(* IEC 61131-3 sources: CodesysTest/export (part 3) *)

(* ---- FB_PneuBagOpenFingersWithSensorsOLD.st ---- *)
{attribute 'FBVisuCreator'}
FUNCTION_BLOCK FB_PneuBagOpenFingersWithSensorsOLD EXTENDS FB_BaseBagOpenFingersOLD
VAR_INPUT
	fingerActuators : IUpDown;
END_VAR
VAR_OUTPUT
END_VAR
VAR
	bagMissingLeft : BOOL;
	bagMissingRight : BOOL;
	simBagPresentLeft : FB_SimulatedFeedbackPhysicalInput(name := CONCAT(_prefix,'Bag Present Left')) := (minDelay := 20, maxDelay := 30);
	simBagPresentRight : FB_SimulatedFeedbackPhysicalInput(name := CONCAT(_prefix,'Bag Present Right')) := (minDelay := 20, maxDelay := 30);
END_VAR
VAR_IN_OUT
	BagPresentSensorLeft : FB_PhysicalDigitalInput;
	BagPresentSensorRight : FB_PhysicalDigitalInput;
END_VAR

SUPER^();
IF simulateIO THEN
	//RotateDownCMD.simulate := RotateUpCMD.simulate := BagPresentSensorLeft.simulate := BagPresentSensorRight.simulate := TRUE;
	BagPresentSensorLeft.simulate := BagPresentSensorRight.simulate := TRUE;
	EnableSimulation(device := fingerActuators, enableSim := TRUE);
END_IF

simBagPresentLeft(in := fingerActuators.DownAsserted,
					simFeedbackFault := UN00_Globals.simFaults.failedToGrabBagLeftFinger OR UN00_Globals.simFaults.failedToGrabBagBothFingers,
					inputToSimulate := BagPresentSensorLeft);
simBagPresentRight(in := fingerActuators.DownAsserted,
					simFeedbackFault := UN00_Globals.simFaults.failedToGrabBagRightFinger OR UN00_Globals.simFaults.failedToGrabBagBothFingers,
					inputToSimulate := BagPresentSensorRight);

bagMissingLeft := NOT BagPresentSensorLeft.Active;
bagMissingRight := NOT BagPresentSensorRight.Active;

IF delayToGrab.Q THEN
	fingerActuators.MoveDown();
	_bagMissed := (bagMissingLeft OR bagMissingRight) AND delayToCheckBagPresent.Q;
	_bagGrabbed := (BagPresentSensorLeft.Active AND BagPresentSensorRight.Active) AND delayToCheckBagPresent.Q;
	//_grabBagRequest := FALSE;
END_IF

IF _releaseBagRequest THEN
	fingerActuators.MoveUp();
	_releaseBagRequest := FALSE;
	_grabBagRequest := FALSE;
END_IF

METHOD RemovePower
VAR_INPUT
END_VAR

SUPER^.RemovePower();

// Try to exhaust the BOF actuators, if the solenoid valve doesn't have that ability then move the fingers up
IF NOT ExhaustIfPossible(fingerActuators) THEN
	fingerActuators.MoveUp();
END_IF

{attribute 'FBVisuCreator'}
FUNCTION_BLOCK FB_PneuBagOpenFingersWithSensorsOLD EXTENDS FB_BaseBagOpenFingersOLD
VAR_INPUT
	fingerActuators : IUpDown;
END_VAR
VAR_OUTPUT
END_VAR
VAR
	bagMissingLeft : BOOL;
	bagMissingRight : BOOL;
	simBagPresentLeft : FB_SimulatedFeedbackPhysicalInput(name := CONCAT(_prefix,'Bag Present Left')) := (minDelay := 20, maxDelay := 30);
	simBagPresentRight : FB_SimulatedFeedbackPhysicalInput(name := CONCAT(_prefix,'Bag Present Right')) := (minDelay := 20, maxDelay := 30);
END_VAR
VAR_IN_OUT
	BagPresentSensorLeft : FB_PhysicalDigitalInput;
	BagPresentSensorRight : FB_PhysicalDigitalInput;
END_VAR

SUPER^();
IF simulateIO THEN
	//RotateDownCMD.simulate := RotateUpCMD.simulate := BagPresentSensorLeft.simulate := BagPresentSensorRight.simulate := TRUE;
	BagPresentSensorLeft.simulate := BagPresentSensorRight.simulate := TRUE;
	EnableSimulation(device := fingerActuators, enableSim := TRUE);
END_IF

simBagPresentLeft(in := fingerActuators.DownAsserted,
					simFeedbackFault := UN00_Globals.simFaults.failedToGrabBagLeftFinger OR UN00_Globals.simFaults.failedToGrabBagBothFingers,
					inputToSimulate := BagPresentSensorLeft);
simBagPresentRight(in := fingerActuators.DownAsserted,
					simFeedbackFault := UN00_Globals.simFaults.failedToGrabBagRightFinger OR UN00_Globals.simFaults.failedToGrabBagBothFingers,
					inputToSimulate := BagPresentSensorRight);

bagMissingLeft := NOT BagPresentSensorLeft.Active;
bagMissingRight := NOT BagPresentSensorRight.Active;

IF delayToGrab.Q THEN
	fingerActuators.MoveDown();
	_bagMissed := (bagMissingLeft OR bagMissingRight) AND delayToCheckBagPresent.Q;
	_bagGrabbed := (BagPresentSensorLeft.Active AND BagPresentSensorRight.Active) AND delayToCheckBagPresent.Q;
	//_grabBagRequest := FALSE;
END_IF

IF _releaseBagRequest THEN
	fingerActuators.MoveUp();
	_releaseBagRequest := FALSE;
	_grabBagRequest := FALSE;
END_IF

METHOD RemovePower
VAR_INPUT
END_VAR

SUPER^.RemovePower();

// Try to exhaust the BOF actuators, if the solenoid valve doesn't have that ability then move the fingers up
IF NOT ExhaustIfPossible(fingerActuators) THEN
	fingerActuators.MoveUp();
END_IF

(* ---- FB_PneumaticActuator.st ---- *)
FUNCTION_BLOCK FB_PneumaticActuator EXTENDS FB_SolenoidValve IMPLEMENTS ICylinder
VAR_INPUT

END_VAR
VAR_OUTPUT
END_VAR
VAR
	_extendAsserted : BOOL;
	_isExtended : BOOL;
	_retractAsserted : BOOL;
	_isRetracted : BOOL;
END_VAR

PROPERTY ExtendAsserted : BOOL

PROPERTY IsExtended : BOOL

PROPERTY IsRetracted : BOOL

PROPERTY RetractAsserted : BOOL

METHOD Extend

_extendAsserted := TRUE;
_retractAsserted := FALSE;

METHOD Retract

_extendAsserted := FALSE;
_retractAsserted := TRUE;

FUNCTION_BLOCK FB_PneumaticActuator EXTENDS FB_SolenoidValve IMPLEMENTS ICylinder
VAR_INPUT

END_VAR
VAR_OUTPUT
END_VAR
VAR
	_extendAsserted : BOOL;
	_isExtended : BOOL;
	_retractAsserted : BOOL;
	_isRetracted : BOOL;
END_VAR

PROPERTY ExtendAsserted : BOOL

PROPERTY IsExtended : BOOL

PROPERTY IsRetracted : BOOL

PROPERTY RetractAsserted : BOOL

METHOD Extend

_extendAsserted := TRUE;
_retractAsserted := FALSE;

METHOD Retract

_extendAsserted := FALSE;
_retractAsserted := TRUE;

(* ---- FB_PneumaticActuator_UnitTests.st ---- *)
(*
*)
{attribute 'test' := 'multitest'}
{attribute 'testcasename':='Base Pneumatic Actuator/Valve'}
{attribute 'testcategory':='Solenoids'}
{attribute 'testcasetimeout':='15000'}
FUNCTION_BLOCK FB_PneumaticActuator_UnitTests EXTENDS CBM.EtrigA
VAR_INPUT
	xGetTestInfo : BOOL;
    diTestCaseIndex : DINT;
END_VAR
VAR_OUTPUT
    sTestCaseName : STRING;
	sTestCaseCategories : STRING;
    diTestCaseCount : DINT;
    diTestCaseTimeout : DINT;
    sInfo : STRING;
	eError : UnitTestErrors;
    sError : STRING;
    eFailureMode : TM.FAILUREMODE;
END_VAR
VAR
	testee : FB_PneumaticActuator(name := 'Unit Test Actuator');
END_VAR
SUPER^();

{attribute 'hide'}
METHOD prvAbort : BOOL

SUPER^.prvAbort();

xAbortInProgress := FALSE;

{attribute 'hide'}
METHOD prvCyclicAction : BOOL

SUPER^.prvCyclicAction();
THIS^.diTestCaseCount := 3;

CASE diTestCaseIndex OF
    0: // Test Case #0
        IF THIS^.xGetTestInfo THEN
            THIS^.sTestCaseName := 'Step 1: Test Initialzed No State';
            THIS^.sTestCaseCategories := 'Solenoids';
            THIS^.diTestCaseTimeout := 3000;
			xDone := TRUE;
		ELSE
			IF NOT testee.ExtendAsserted
				AND NOT testee.RetractAsserted
				AND NOT testee.IsExtended
				AND NOT testee.IsRetracted
				THEN
				 xDone := TRUE;
			ELSE
				THIS^.sError := 'Initialzed with state (Extended or Retracted)';
				xError := TRUE;
				eError := UnitTestErrors.Failure;
            	eFailureMode := TM.FAILUREMODE.AbortTestCase;
                iError := 1;
			END_IF
        END_IF
    1: // Test Case #1
        IF THIS^.xGetTestInfo THEN
            THIS^.sTestCaseName := 'Step 2: Extend Cylinder';
            THIS^.sTestCaseCategories := 'Solenoids';
            THIS^.diTestCaseTimeout := 3000;
            xDone := TRUE;
		ELSE
			testee.Extend();
			testee.IsExtended := TRUE;
			IF testee.ExtendAsserted
				AND testee.IsExtended
				AND NOT testee.RetractAsserted
				AND NOT testee.IsRetracted
				THEN
				 xDone := TRUE;
			ELSE
				THIS^.sError := 'Failed to extend';
				xError := TRUE;
				eError := UnitTestErrors.Failure;
            	eFailureMode := TM.FAILUREMODE.AbortTestCase;
                iError := 2;
			END_IF
       END_IF

	2:	//
		IF THIS^.xGetTestInfo THEN
            THIS^.sTestCaseName := 'Step 3: Retract Cylinder';
            THIS^.sTestCaseCategories := 'Solenoids';
            THIS^.diTestCaseTimeout := 3000;
            xDone := TRUE;
		ELSE
			testee.Retract();
			testee.IsRetracted := TRUE;
			testee.IsExtended := FALSE;
			IF NOT testee.ExtendAsserted
				AND NOT testee.IsExtended
				AND testee.RetractAsserted
				AND testee.IsRetracted
				THEN
				 xDone := TRUE;
			ELSE
				THIS^.sError := 'Failed to retract';
				xError := TRUE;
				eError := UnitTestErrors.Failure;
            	eFailureMode := TM.FAILUREMODE.AbortTestCase;
                iError := 3;
			END_IF
       END_IF
    ELSE
        IF THIS^.diTestCaseIndex < 0 THEN
            THIS^.diTestCaseCount := 3;
            xDone := TRUE;
        ELSE
            THIS^.sInfo := 'Invalid test case index';
            eError := UnitTestErrors.Failure;
			xError := TRUE;
        END_IF
END_CASE

{attribute 'hide'}
METHOD prvResetOutputs : BOOL

SUPER^.prvResetOutputs();

sTestCaseName := '';
sTestCaseCategories := '';
diTestCaseCount := 0;
diTestCaseTimeout := 0;
sInfo := '';
sError := '';
eFailureMode := TM.FAILUREMODE.AbortTestCase;

{attribute 'hide'}
METHOD prvStart : BOOL

SUPER^.prvStart();

(*
*)
{attribute 'test' := 'multitest'}
{attribute 'testcasename':='Base Pneumatic Actuator/Valve'}
{attribute 'testcategory':='Solenoids'}
{attribute 'testcasetimeout':='15000'}
FUNCTION_BLOCK FB_PneumaticActuator_UnitTests EXTENDS CBM.EtrigA
VAR_INPUT
	xGetTestInfo : BOOL;
    diTestCaseIndex : DINT;
END_VAR
VAR_OUTPUT
    sTestCaseName : STRING;
	sTestCaseCategories : STRING;
    diTestCaseCount : DINT;
    diTestCaseTimeout : DINT;
    sInfo : STRING;
	eError : UnitTestErrors;
    sError : STRING;
    eFailureMode : TM.FAILUREMODE;
END_VAR
VAR
	testee : FB_PneumaticActuator(name := 'Unit Test Actuator');
END_VAR
SUPER^();

{attribute 'hide'}
METHOD prvAbort : BOOL

SUPER^.prvAbort();

xAbortInProgress := FALSE;

{attribute 'hide'}
METHOD prvCyclicAction : BOOL

SUPER^.prvCyclicAction();
THIS^.diTestCaseCount := 3;

CASE diTestCaseIndex OF
    0: // Test Case #0
        IF THIS^.xGetTestInfo THEN
            THIS^.sTestCaseName := 'Step 1: Test Initialzed No State';
            THIS^.sTestCaseCategories := 'Solenoids';
            THIS^.diTestCaseTimeout := 3000;
			xDone := TRUE;
		ELSE
			IF NOT testee.ExtendAsserted
				AND NOT testee.RetractAsserted
				AND NOT testee.IsExtended
				AND NOT testee.IsRetracted
				THEN
				 xDone := TRUE;
			ELSE
				THIS^.sError := 'Initialzed with state (Extended or Retracted)';
				xError := TRUE;
				eError := UnitTestErrors.Failure;
            	eFailureMode := TM.FAILUREMODE.AbortTestCase;
                iError := 1;
			END_IF
        END_IF
    1: // Test Case #1
        IF THIS^.xGetTestInfo THEN
            THIS^.sTestCaseName := 'Step 2: Extend Cylinder';
            THIS^.sTestCaseCategories := 'Solenoids';
            THIS^.diTestCaseTimeout := 3000;
            xDone := TRUE;
		ELSE
			testee.Extend();
			testee.IsExtended := TRUE;
			IF testee.ExtendAsserted
				AND testee.IsExtended
				AND NOT testee.RetractAsserted
				AND NOT testee.IsRetracted
				THEN
				 xDone := TRUE;
			ELSE
				THIS^.sError := 'Failed to extend';
				xError := TRUE;
				eError := UnitTestErrors.Failure;
            	eFailureMode := TM.FAILUREMODE.AbortTestCase;
                iError := 2;
			END_IF
       END_IF

	2:	//
		IF THIS^.xGetTestInfo THEN
            THIS^.sTestCaseName := 'Step 3: Retract Cylinder';
            THIS^.sTestCaseCategories := 'Solenoids';
            THIS^.diTestCaseTimeout := 3000;
            xDone := TRUE;
		ELSE
			testee.Retract();
			testee.IsRetracted := TRUE;
			testee.IsExtended := FALSE;
			IF NOT testee.ExtendAsserted
				AND NOT testee.IsExtended
				AND testee.RetractAsserted
				AND testee.IsRetracted
				THEN
				 xDone := TRUE;
			ELSE
				THIS^.sError := 'Failed to retract';
				xError := TRUE;
				eError := UnitTestErrors.Failure;
            	eFailureMode := TM.FAILUREMODE.AbortTestCase;
                iError := 3;
			END_IF
       END_IF
    ELSE
        IF THIS^.diTestCaseIndex < 0 THEN
            THIS^.diTestCaseCount := 3;
            xDone := TRUE;
        ELSE
            THIS^.sInfo := 'Invalid test case index';
            eError := UnitTestErrors.Failure;
			xError := TRUE;
        END_IF
END_CASE

{attribute 'hide'}
METHOD prvResetOutputs : BOOL

SUPER^.prvResetOutputs();

sTestCaseName := '';
sTestCaseCategories := '';
diTestCaseCount := 0;
diTestCaseTimeout := 0;
sInfo := '';
sError := '';
eFailureMode := TM.FAILUREMODE.AbortTestCase;

{attribute 'hide'}
METHOD prvStart : BOOL

SUPER^.prvStart();

(* ---- FB_PneumaticSealer.st ---- *)
FUNCTION_BLOCK FINAL FB_PneumaticSealer EXTENDS FB_BasicSealer
VAR_INPUT
	cylinder : ICylinder;
END_VAR
VAR_OUTPUT
END_VAR
VAR

END_VAR

SUPER^();

EnableSimulation(cylinder,simulateIO);

IF sealActive THEN
	cylinder.Extend();
ELSE
	cylinder.Retract();
END_IF

{attribute 'monitoring' := 'variable'}
PROPERTY SealComplete : BOOL

METHOD BeginSealing

_beginSealing := TRUE;
sealTimer.IN := FALSE;
_sealComplete := FALSE;

FUNCTION_BLOCK FINAL FB_PneumaticSealer EXTENDS FB_BasicSealer
VAR_INPUT
	cylinder : ICylinder;
END_VAR
VAR_OUTPUT
END_VAR
VAR

END_VAR

SUPER^();

EnableSimulation(cylinder,simulateIO);

IF sealActive THEN
	cylinder.Extend();
ELSE
	cylinder.Retract();
END_IF

{attribute 'monitoring' := 'variable'}
PROPERTY SealComplete : BOOL

METHOD BeginSealing

_beginSealing := TRUE;
sealTimer.IN := FALSE;
_sealComplete := FALSE;

(* ---- FB_PneumaticVacuumCups.st ---- *)
FUNCTION_BLOCK FB_PneumaticVacuumCups EXTENDS FB_BaseComponent IMPLEMENTS IVacuumBagOpen
VAR_INPUT

END_VAR
VAR_OUTPUT

END_VAR
VAR
	_vacuumOn : BOOL;
END_VAR
VAR_IN_OUT
	vacGenerator : FB_VacuumGenerator;
END_VAR
SUPER^();

{attribute 'monitoring' := 'variable'}
PROPERTY VacuumOn : BOOL

METHOD StartVacuum

vacGenerator.GeneratorsOn();
_vacuumOn := TRUE;

METHOD StopVacuum

vacGenerator.GeneratorsOff();
_vacuumOn := FALSE;

(* ---- FB_PneumaticVacuumCups_UnitTests.st ---- *)
{attribute 'test' := 'multitest'}
{attribute 'testcasename':='Pneumatic Vacuum Cups'}
{attribute 'testcategory':='Machine Components'}
{attribute 'testcasetimeout':='15000'}

FUNCTION_BLOCK FB_PneumaticVacuumCups_UnitTests EXTENDS CBM.EtrigA
VAR_INPUT
	xGetTestInfo : BOOL;
    diTestCaseIndex : DINT;
END_VAR
VAR_OUTPUT
    sTestCaseName : STRING;
	sTestCaseCategories : STRING;
    diTestCaseCount : DINT;
    diTestCaseTimeout : DINT;
    sInfo : STRING;
	eError : UnitTestErrors;
    sError : STRING;
    eFailureMode : TM.FAILUREMODE;
END_VAR
VAR
	testVacGenerator : FB_VacuumGenerator(name := 'Test Vac Generator');
	testee : FB_PneumaticVacuumCups(name := 'Test Pneumatic Vac Cups');
END_VAR
SUPER^();
testVacGenerator();
testee(vacGenerator := testVacGenerator);

{attribute 'hide'}
METHOD prvAbort : BOOL

SUPER^.prvAbort();

xAbortInProgress := FALSE;

{attribute 'hide'}
METHOD prvCyclicAction : BOOL

SUPER^.prvCyclicAction();

CASE diTestCaseIndex OF
    0: 	IF THIS^.xGetTestInfo THEN
            THIS^.sTestCaseName := 'Step 1: Check Vacuum Is Off On Initialze';
            THIS^.sTestCaseCategories := 'General';
            THIS^.diTestCaseTimeout := 3000;
			xDone := TRUE;
		ELSE
			IF testee.VacuumOn = FALSE THEN
				 xDone := TRUE;
			ELSE
				THIS^.sError := 'Vacuum On, should be off on initialize';
				xError := TRUE;
				eError := UnitTestErrors.Failure;
            	eFailureMode := TM.FAILUREMODE.AbortTestCase;
                iError := 1;
			END_IF
        END_IF
    1: 	IF THIS^.xGetTestInfo THEN
            THIS^.sTestCaseName := 'Step 2: Start Vacuum';
            THIS^.sTestCaseCategories := 'General';
            THIS^.diTestCaseTimeout := 3000;
			xDone := TRUE;
		ELSE
			testee.StartVacuum();
			IF testee.VacuumOn AND testVacGenerator.Solenoid0Asserted THEN
				 xDone := TRUE;
			ELSE
				THIS^.sError := 'Vacuum Off, should be on';
				xError := TRUE;
				eError := UnitTestErrors.Failure;
            	eFailureMode := TM.FAILUREMODE.AbortTestCase;
                iError := 1;
			END_IF
        END_IF

	2: 	IF THIS^.xGetTestInfo THEN
            THIS^.sTestCaseName := 'Step 3: Stop Vacuum';
            THIS^.sTestCaseCategories := 'General';
            THIS^.diTestCaseTimeout := 3000;
			xDone := TRUE;
		ELSE
			testee.StopVacuum();
			IF NOT testee.VacuumOn AND NOT testVacGenerator.Solenoid0Asserted THEN
				 xDone := TRUE;
			ELSE
				THIS^.sError := 'Vacumm On, should be off';
				xError := TRUE;
				eError := UnitTestErrors.Failure;
            	eFailureMode := TM.FAILUREMODE.AbortTestCase;
                iError := 1;
			END_IF
        END_IF

   	3: 	IF THIS^.xGetTestInfo THEN
            THIS^.sTestCaseName := 'Step 4: ';
            THIS^.sTestCaseCategories := 'General';
            THIS^.diTestCaseTimeout := 3000;
			xDone := TRUE;
		ELSE
			(*TEST SOMETHING HERE*)
			IF (*CONNDITION*) FALSE THEN
				 xDone := TRUE;
			ELSE
				THIS^.sError := '';
				xError := TRUE;
				eError := UnitTestErrors.Failure;
            	eFailureMode := TM.FAILUREMODE.AbortTestCase;
                iError := 1;
			END_IF
        END_IF

	4: 	IF THIS^.xGetTestInfo THEN
            THIS^.sTestCaseName := 'Step 5: ';
            THIS^.sTestCaseCategories := 'General';
            THIS^.diTestCaseTimeout := 3000;
			xDone := TRUE;
		ELSE
			(*TEST SOMETHING HERE*)
			IF (*CONNDITION*) FALSE THEN
				 xDone := TRUE;
			ELSE
				THIS^.sError := '';
				xError := TRUE;
				eError := UnitTestErrors.Failure;
            	eFailureMode := TM.FAILUREMODE.AbortTestCase;
                iError := 1;
			END_IF
        END_IF

	5: 	IF THIS^.xGetTestInfo THEN
            THIS^.sTestCaseName := 'Step 6: ';
            THIS^.sTestCaseCategories := 'General';
            THIS^.diTestCaseTimeout := 3000;
			xDone := TRUE;
		ELSE
			(*TEST SOMETHING HERE*)
			IF (*CONNDITION*) FALSE THEN
				 xDone := TRUE;
			ELSE
				THIS^.sError := '';
				xError := TRUE;
				eError := UnitTestErrors.Failure;
            	eFailureMode := TM.FAILUREMODE.AbortTestCase;
                iError := 1;
			END_IF
        END_IF

	6: 	IF THIS^.xGetTestInfo THEN
            THIS^.sTestCaseName := 'Step 7: ';
            THIS^.sTestCaseCategories := 'General';
            THIS^.diTestCaseTimeout := 3000;
			xDone := TRUE;
		ELSE
			(*TEST SOMETHING HERE*)
			IF (*CONNDITION*) FALSE THEN
				 xDone := TRUE;
			ELSE
				THIS^.sError := '';
				xError := TRUE;
				eError := UnitTestErrors.Failure;
            	eFailureMode := TM.FAILUREMODE.AbortTestCase;
                iError := 1;
			END_IF
        END_IF
    ELSE
        IF THIS^.diTestCaseIndex < 0 THEN
            THIS^.diTestCaseCount := 3;
            xDone := TRUE;
        ELSE
            THIS^.sInfo := 'Invalid test case index';
            eError := UnitTestErrors.Failure;
			xError := TRUE;
        END_IF
END_CASE

{attribute 'hide'}
METHOD prvResetOutputs : BOOL

SUPER^.prvResetOutputs();

sTestCaseName := '';
sTestCaseCategories := '';
diTestCaseCount := 0;
diTestCaseTimeout := 0;
sInfo := '';
sError := '';
eFailureMode := TM.FAILUREMODE.AbortTestCase;

{attribute 'hide'}
METHOD prvStart : BOOL

{attribute 'test' := 'multitest'}
{attribute 'testcasename':='Pneumatic Vacuum Cups'}
{attribute 'testcategory':='Machine Components'}
{attribute 'testcasetimeout':='15000'}

FUNCTION_BLOCK FB_PneumaticVacuumCups_UnitTests EXTENDS CBM.EtrigA
VAR_INPUT
	xGetTestInfo : BOOL;
    diTestCaseIndex : DINT;
END_VAR
VAR_OUTPUT
    sTestCaseName : STRING;
	sTestCaseCategories : STRING;
    diTestCaseCount : DINT;
    diTestCaseTimeout : DINT;
    sInfo : STRING;
	eError : UnitTestErrors;
    sError : STRING;
    eFailureMode : TM.FAILUREMODE;
END_VAR
VAR
	testVacGenerator : FB_VacuumGenerator(name := 'Test Vac Generator');
	testee : FB_PneumaticVacuumCups(name := 'Test Pneumatic Vac Cups');
END_VAR
SUPER^();
testVacGenerator();
testee(vacGenerator := testVacGenerator);

{attribute 'hide'}
METHOD prvAbort : BOOL

SUPER^.prvAbort();

xAbortInProgress := FALSE;

{attribute 'hide'}
METHOD prvCyclicAction : BOOL

SUPER^.prvCyclicAction();

CASE diTestCaseIndex OF
    0: 	IF THIS^.xGetTestInfo THEN
            THIS^.sTestCaseName := 'Step 1: Check Vacuum Is Off On Initialze';
            THIS^.sTestCaseCategories := 'General';
            THIS^.diTestCaseTimeout := 3000;
			xDone := TRUE;
		ELSE
			IF testee.VacuumOn = FALSE THEN
				 xDone := TRUE;
			ELSE
				THIS^.sError := 'Vacuum On, should be off on initialize';
				xError := TRUE;
				eError := UnitTestErrors.Failure;
            	eFailureMode := TM.FAILUREMODE.AbortTestCase;
                iError := 1;
			END_IF
        END_IF
    1: 	IF THIS^.xGetTestInfo THEN
            THIS^.sTestCaseName := 'Step 2: Start Vacuum';
            THIS^.sTestCaseCategories := 'General';
            THIS^.diTestCaseTimeout := 3000;
			xDone := TRUE;
		ELSE
			testee.StartVacuum();
			IF testee.VacuumOn AND testVacGenerator.Solenoid0Asserted THEN
				 xDone := TRUE;
			ELSE
				THIS^.sError := 'Vacuum Off, should be on';
				xError := TRUE;
				eError := UnitTestErrors.Failure;
            	eFailureMode := TM.FAILUREMODE.AbortTestCase;
                iError := 1;
			END_IF
        END_IF

	2: 	IF THIS^.xGetTestInfo THEN
            THIS^.sTestCaseName := 'Step 3: Stop Vacuum';
            THIS^.sTestCaseCategories := 'General';
            THIS^.diTestCaseTimeout := 3000;
			xDone := TRUE;
		ELSE
			testee.StopVacuum();
			IF NOT testee.VacuumOn AND NOT testVacGenerator.Solenoid0Asserted THEN
				 xDone := TRUE;
			ELSE
				THIS^.sError := 'Vacumm On, should be off';
				xError := TRUE;
				eError := UnitTestErrors.Failure;
            	eFailureMode := TM.FAILUREMODE.AbortTestCase;
                iError := 1;
			END_IF
        END_IF

   	3: 	IF THIS^.xGetTestInfo THEN
            THIS^.sTestCaseName := 'Step 4: ';
            THIS^.sTestCaseCategories := 'General';
            THIS^.diTestCaseTimeout := 3000;
			xDone := TRUE;
		ELSE
			(*TEST SOMETHING HERE*)
			IF (*CONNDITION*) FALSE THEN
				 xDone := TRUE;
			ELSE
				THIS^.sError := '';
				xError := TRUE;
				eError := UnitTestErrors.Failure;
            	eFailureMode := TM.FAILUREMODE.AbortTestCase;
                iError := 1;
			END_IF
        END_IF

	4: 	IF THIS^.xGetTestInfo THEN
            THIS^.sTestCaseName := 'Step 5: ';
            THIS^.sTestCaseCategories := 'General';
            THIS^.diTestCaseTimeout := 3000;
			xDone := TRUE;
		ELSE
			(*TEST SOMETHING HERE*)
			IF (*CONNDITION*) FALSE THEN
				 xDone := TRUE;
			ELSE
				THIS^.sError := '';
				xError := TRUE;
				eError := UnitTestErrors.Failure;
            	eFailureMode := TM.FAILUREMODE.AbortTestCase;
                iError := 1;
			END_IF
        END_IF

	5: 	IF THIS^.xGetTestInfo THEN
            THIS^.sTestCaseName := 'Step 6: ';
            THIS^.sTestCaseCategories := 'General';
            THIS^.diTestCaseTimeout := 3000;
			xDone := TRUE;
		ELSE
			(*TEST SOMETHING HERE*)
			IF (*CONNDITION*) FALSE THEN
				 xDone := TRUE;
			ELSE
				THIS^.sError := '';
				xError := TRUE;
				eError := UnitTestErrors.Failure;
            	eFailureMode := TM.FAILUREMODE.AbortTestCase;
                iError := 1;
			END_IF
        END_IF

	6: 	IF THIS^.xGetTestInfo THEN
            THIS^.sTestCaseName := 'Step 7: ';
            THIS^.sTestCaseCategories := 'General';
            THIS^.diTestCaseTimeout := 3000;
			xDone := TRUE;
		ELSE
			(*TEST SOMETHING HERE*)
			IF (*CONNDITION*) FALSE THEN
				 xDone := TRUE;
			ELSE
				THIS^.sError := '';
				xError := TRUE;
				eError := UnitTestErrors.Failure;
            	eFailureMode := TM.FAILUREMODE.AbortTestCase;
                iError := 1;
			END_IF
        END_IF
    ELSE
        IF THIS^.diTestCaseIndex < 0 THEN
            THIS^.diTestCaseCount := 3;
            xDone := TRUE;
        ELSE
            THIS^.sInfo := 'Invalid test case index';
            eError := UnitTestErrors.Failure;
			xError := TRUE;
        END_IF
END_CASE

{attribute 'hide'}
METHOD prvResetOutputs : BOOL

SUPER^.prvResetOutputs();

sTestCaseName := '';
sTestCaseCategories := '';
diTestCaseCount := 0;
diTestCaseTimeout := 0;
sInfo := '';
sError := '';
eFailureMode := TM.FAILUREMODE.AbortTestCase;

{attribute 'hide'}
METHOD prvStart : BOOL

(* ---- FB_PneumaticVerticalActuator.st ---- *)
FUNCTION_BLOCK FB_PneumaticVerticalActuator EXTENDS FB_PneumaticActuator IMPLEMENTS IUpDown
VAR_INPUT
	cylinder : ICylinder;
END_VAR
VAR_OUTPUT
END_VAR
VAR
END_VAR
VAR_IN_OUT
END_VAR

//	Function Block: FB_PneumaticVerticalActuator
//	Description: Wrapper for a cylinder with Up/Down substitiuted for Extend/Retract
//
//
//	Usage:
//
//	Created by: Ben Hess
//	Created Date: 6-27-2019

EnableSimulation(cylinder, _simulateActive);

PROPERTY UpAsserted : BOOL

PROPERTY DownAsserted : BOOL

PROPERTY IsDown : BOOL

PROPERTY IsUp : BOOL

METHOD MoveDown

cylinder.Extend();

METHOD MoveUp

cylinder.Retract();

(* ---- FB_PneuPBarWithAdjPass.st ---- *)
FUNCTION_BLOCK FB_PneuPBarWithAdjPass EXTENDS FB_BaseComponent IMPLEMENTS IPressureBar, IHomable, IPostHomeMove
VAR_INPUT
	simulateIO : BOOL;												// Simulate all I/O for testing
	passthroughMotor : REFERENCE TO Sharp_Motion.Axis_REF;			// The motor axis for the passthrough
	ptVelo : REAL := 0.5;											// Passthrough Motor Velocity
	ptAccel : REAL := 10.0;											// Passthrough Motor Acceleration
	ptDecel : REAL := 1.0;											// Passthrough Motor Deceleration
	homeTimeoutSetting : TIME := T#20S;								// Timeout for homing attempt
	passthroughSetting : REAL := 8.0;
	cylinder : ICylinder;
END_VAR
VAR_OUTPUT
	failedToClose : FB_Fault(name := CONCAT(_prefix, 'Failed to Close'));
	failedToOpen : FB_Fault(name := CONCAT(_prefix, 'Failed to Open'));
	failedToHome : FB_Fault(name := CONCAT(_prefix, 'Failed to Home'));
	pressureBarObstructed : FB_Fault(name := CONCAT(_prefix, 'Obstructed'));
	motorFault : FB_Fault(name := CONCAT(_prefix, 'Motor Fault'));
	failedToMovePassthrough : FB_Fault(name := CONCAT(_prefix, 'Failed to Move Passthrough'));
	actualPassthrough : REAL := 8.0;								// Current Passthrough Opening
	//CloseSolenoid : FB_PhysicalDigitalOutput(name := CONCAT(_prefix, 'Close Solenoid'));
	//OpenSolenoid : FB_PhysicalDigitalOutput(name := CONCAT(_prefix, 'Open Solenoid'));
END_VAR
VAR
	simClose : FB_SimulatedFeedbackPhysicalInput(name := CONCAT(_prefix,'Move In')) := (minDelay := 20, maxDelay := 60);
	simOpen : FB_SimulatedFeedbackPhysicalInput(name := CONCAT(_prefix,'Move Out')) := (minDelay := 20, maxDelay := 60);
	MC_HomePassthrough : Sharp_Motion.MC_Home;
	MC_MovePassthrough : Sharp_Motion.MC_MoveAbsolute;
	MC_ResetPassthoughMotor : Sharp_Motion.MC_Reset;
	MC_HaltPasstroughMotor : Sharp_Motion.MC_Halt;
	_homeNow : BOOL;
	_movePassthroughNow : BOOL;
	_isFullyClosed : BOOL;
	_isFullyOpen : BOOL;
	adjustablePassthroughState : INT;
	homeTimeout : Standard.TON;
	movePassthroughTimeout : Standard.TON;
	failedToCloseTimer : Standard.TON;
	failedToOpenTimer : Standard.TON;
	faultTime : TIME := T#5S;
END_VAR
VAR_IN_OUT
	PressureBarClosedSensor : FB_PhysicalDigitalInput;
	PressureBarOpenSensor : FB_PhysicalDigitalInput;
	ObstructionSensor : FB_PhysicalDigitalInput;
END_VAR
//	Function Block: FB_PneuPBarWithAdjPass()
//	Description: Pneumatic pressure bar with adjustable passthrough - passthrough adjustment is done with motor
//
//	Created by: Ben Hess
//	Created Date: Tuesday, May 14th, 2019

SUPER^();

{region "Axis Setup"}
// Setup of Motion Commands for passthrough motor axis
MC_HomePassthrough(Axis := passthroughMotor);
MC_MovePassthrough(Axis := passthroughMotor);
MC_ResetPassthoughMotor(Axis := passthroughMotor);
MC_HaltPasstroughMotor(Axis := passthroughMotor);
{endregion}

{region "Timers"}
// If homing not complete within reasonable time, error out
homeTimeout(PT := homeTimeoutSetting);
// If passthrough doesn't reach setpoint in reasonable time, error out
movePassthroughTimeout();
{endregion}

{region "I/O and Fault Setup"}
// Passthrough position is based on reported motor position
actualPassthrough := passthroughMotor.ActPos;

// Setup simulation of I/O and faults for testing
simClose(in := cylinder.RetractAsserted, simFeedbackFault := UN00_Globals.simFaults.pressureBarFailedToMoveIn, inputToSimulate := PressureBarClosedSensor);
simOpen(in := cylinder.ExtendAsserted, simFeedbackFault := UN00_Globals.simFaults.pressureBarFailedToMoveOut, inputToSimulate := PressureBarOpenSensor);
ObstructionSensor.simulate := PressureBarClosedSensor.simulate := PressureBarOpenSensor.simulate := simulateIO;
ObstructionSensor.simValue := NOT UN00_Globals.simFaults.pressureBarObstucted;
EnableSimulation(device := cylinder, enableSim := simulateIO);

_isFullyClosed := PressureBarClosedSensor.Active;
_isFullyOpen := PressureBarOpenSensor.Active;

// Failed to reach sensor timers
// Exclusively use Close solonoid for Close fail timer since Open slow/low pressure uses both solenoids
failedToCloseTimer(IN := cylinder.RetractAsserted AND NOT _isFullyClosed,
					PT := faultTime,
					Q => failedToClose.faultTrigger);
failedToOpenTimer(IN := cylinder.ExtendAsserted AND NOT _isFullyOpen,
					PT := faultTime,
					Q => failedToOpen.faultTrigger);

// Obstruction fault is normally closed, fail safe.  Fault if collapsable jaw is broken anywhere outside of all the way in or all the way out
pressureBarObstructed.faultTrigger := ObstructionSensor.IsOff AND NOT (_isFullyClosed OR _isFullyOpen)
										OR ObstructionSensor.IsOff AND (_isFullyOpen AND cylinder.RetractAsserted);   // Also fault if broken when we try to close from all the way out
IF passthroughMotor.Error THEN
	motorFault.faultTrigger := TRUE;
	adjustablePassthroughState := 0;
ELSE
	motorFault.faultTrigger := FALSE;
END_IF
{endregion}

IF _reset THEN
	adjustablePassthroughState := 100;
	IF passthroughMotor.Error THEN
		MC_ResetPassthoughMotor.Execute := TRUE;
	END_IF
	_movePassthroughNow := FALSE;
	movePassthroughTimeout.IN := FALSE;
	_reset := FALSE;
END_IF

CASE adjustablePassthroughState OF

	0:  // Idle State.
		MC_ResetPassthoughMotor.Execute := FALSE;
		IF passthroughMotor.HomingDone
			AND NOT failedToClose.Active
			AND NOT failedToOpen.Active
			AND NOT failedToHome.Active
			AND NOT pressureBarObstructed.Active
			AND NOT motorFault.Active
			AND NOT failedToMovePassthrough.Active
			AND InDesiredPosition
		THEN
			_ready := TRUE;
		ELSE
			_ready := FALSE;
		END_IF

		IF _homeNow AND NOT passthroughMotor.HomingDone THEN
			MC_HomePassthrough.Execute := TRUE;
			OpenLowPressure();
			_homeNow := FALSE;
			adjustablePassthroughState := 1;
		ELSIF _homeNow AND passthroughMotor.HomingDone THEN
			_homeNow := FALSE;
		END_IF

		IF _movePassthroughNow AND passthroughMotor.HomingDone THEN
			IF InDesiredPosition THEN
				_movePassthroughNow := FALSE;
				adjustablePassthroughState := 100;
			ELSE
				MC_MovePassthrough.Position := passthroughSetting;
				MC_MovePassthrough.Velocity := ptVelo;
				MC_MovePassthrough.Acceleration := ptAccel;
				MC_MovePassthrough.Deceleration := ptDecel;
				_movePassthroughNow := FALSE;
				OpenLowPressure();

				IF UN00_Globals.simFaults.failedToMovePassthrough THEN
					movePassthroughTimeout.PT := TO_TIME(((ABS(actualPassthrough - passthroughSetting) / ptVelo) * 1000) - 500) ;
				ELSE
					movePassthroughTimeout.PT := TO_TIME(((ABS(actualPassthrough - passthroughSetting) / ptVelo) * 1000) + 2000);
				END_IF

				MC_MovePassthrough.Execute := TRUE;
				adjustablePassthroughState := 2;
			END_IF
		END_IF

	1:	// Homing
		homeTimeout.IN := TRUE;
		IF homeTimeout.Q
			OR MC_HomePassthrough.Error
			OR UN00_Globals.simFaults.pressureBarfailedToHome
		THEN
			failedToHome.Trigger();
			adjustablePassthroughState := 100;
		END_IF
		IF MC_HomePassthrough.Done THEN
			adjustablePassthroughState := 100;
		END_IF

	2:	// Start Moving Passthrough
		movePassthroughTimeout.IN := TRUE;

		IF MC_MovePassthrough.Error OR movePassthroughTimeout.Q THEN
			failedToMovePassthrough.Trigger();
			MC_MovePassthrough.Execute := FALSE;
			MC_HaltPasstroughMotor.Execute := TRUE;
			Exhaust();
			adjustablePassthroughState := 100;
		END_IF

		IF MC_MovePassthrough.Done THEN
			Open();
			MC_MovePassthrough.Execute := FALSE;
			adjustablePassthroughState := 100;
		END_IF

	100:// Cleanup
		MC_HomePassthrough.Execute := FALSE;
		//resetPassthoughMotor.Execute := FALSE;
		MC_MovePassthrough.Execute := FALSE;
		MC_HaltPasstroughMotor.Execute := FALSE;
		homeTimeout.IN := FALSE;
		movePassthroughTimeout.IN := FALSE;
		_homeNow := FALSE;

		adjustablePassthroughState := 0;

END_CASE

METHOD MovePassthrough
VAR_INPUT
	//passthroughSetting : REAL;
END_VAR

//_passthroughSetting := passthroughSetting;
_movePassthroughNow := TRUE;

{attribute 'monitoring' := 'variable'}
PROPERTY IsFullyOpen : BOOL

{attribute 'monitoring' := 'variable'}
PROPERTY IsFullyClosed : BOOL

METHOD Close

simClose.maxDelay := TO_DINT((actualPassthrough / 22.5) * 1000 + 50);
simClose.minDelay := TO_DINT((actualPassthrough / 22.5) * 1000 + 10);

cylinder.Retract();
faultTime := TO_TIME((actualPassthrough / 22.5) * 1000 + 300);

METHOD Open

simOpen.maxDelay := TO_INT((actualPassthrough / 22.5) * 1000 + 50);
simOpen.minDelay := TO_INT((actualPassthrough / 22.5) * 1000 + 10);

cylinder.Extend();
faultTime := TO_TIME((actualPassthrough / 22.5) * 1000 + 300);

METHOD RemovePower
VAR_INPUT
END_VAR

THIS^.Exhaust();
MC_HaltPasstroughMotor.Execute := TRUE;

PROPERTY IsHomed : BOOL

METHOD HomeNow
VAR_INPUT
END_VAR

_homeNow := TRUE;

METHOD OpenLowPressure
VAR_INPUT
END_VAR

simOpen.maxDelay := TO_INT((actualPassthrough / 4) * 1000 + 50);
simOpen.minDelay := TO_INT((actualPassthrough / 4) * 1000 + 10);
simOpen.faultDelay := simClose.maxDelay + 300;

ExtendLPIfPossible(cylinder);
faultTime := TO_TIME((actualPassthrough / 4) * 1000 + 300);

METHOD Exhaust
VAR_INPUT
END_VAR

ExhaustIfPossible(cylinder);

METHOD MoveNow
VAR_INPUT
END_VAR

THIS^.MovePassthrough();

PROPERTY InDesiredPosition : BOOL

FUNCTION_BLOCK FB_PneuPBarWithAdjPass EXTENDS FB_BaseComponent IMPLEMENTS IPressureBar, IHomable, IPostHomeMove
VAR_INPUT
	simulateIO : BOOL;												// Simulate all I/O for testing
	passthroughMotor : REFERENCE TO Sharp_Motion.Axis_REF;			// The motor axis for the passthrough
	ptVelo : REAL := 0.5;											// Passthrough Motor Velocity
	ptAccel : REAL := 10.0;											// Passthrough Motor Acceleration
	ptDecel : REAL := 1.0;											// Passthrough Motor Deceleration
	homeTimeoutSetting : TIME := T#20S;								// Timeout for homing attempt
	passthroughSetting : REAL := 8.0;
	cylinder : ICylinder;
END_VAR
VAR_OUTPUT
	failedToClose : FB_Fault(name := CONCAT(_prefix, 'Failed to Close'));
	failedToOpen : FB_Fault(name := CONCAT(_prefix, 'Failed to Open'));
	failedToHome : FB_Fault(name := CONCAT(_prefix, 'Failed to Home'));
	pressureBarObstructed : FB_Fault(name := CONCAT(_prefix, 'Obstructed'));
	motorFault : FB_Fault(name := CONCAT(_prefix, 'Motor Fault'));
	failedToMovePassthrough : FB_Fault(name := CONCAT(_prefix, 'Failed to Move Passthrough'));
	actualPassthrough : REAL := 8.0;								// Current Passthrough Opening
	//CloseSolenoid : FB_PhysicalDigitalOutput(name := CONCAT(_prefix, 'Close Solenoid'));
	//OpenSolenoid : FB_PhysicalDigitalOutput(name := CONCAT(_prefix, 'Open Solenoid'));
END_VAR
VAR
	simClose : FB_SimulatedFeedbackPhysicalInput(name := CONCAT(_prefix,'Move In')) := (minDelay := 20, maxDelay := 60);
	simOpen : FB_SimulatedFeedbackPhysicalInput(name := CONCAT(_prefix,'Move Out')) := (minDelay := 20, maxDelay := 60);
	MC_HomePassthrough : Sharp_Motion.MC_Home;
	MC_MovePassthrough : Sharp_Motion.MC_MoveAbsolute;
	MC_ResetPassthoughMotor : Sharp_Motion.MC_Reset;
	MC_HaltPasstroughMotor : Sharp_Motion.MC_Halt;
	_homeNow : BOOL;
	_movePassthroughNow : BOOL;
	_isFullyClosed : BOOL;
	_isFullyOpen : BOOL;
	adjustablePassthroughState : INT;
	homeTimeout : Standard.TON;
	movePassthroughTimeout : Standard.TON;
	failedToCloseTimer : Standard.TON;
	failedToOpenTimer : Standard.TON;
	faultTime : TIME := T#5S;
END_VAR
VAR_IN_OUT
	PressureBarClosedSensor : FB_PhysicalDigitalInput;
	PressureBarOpenSensor : FB_PhysicalDigitalInput;
	ObstructionSensor : FB_PhysicalDigitalInput;
END_VAR
//	Function Block: FB_PneuPBarWithAdjPass()
//	Description: Pneumatic pressure bar with adjustable passthrough - passthrough adjustment is done with motor
//
//	Created by: Ben Hess
//	Created Date: Tuesday, May 14th, 2019

SUPER^();

{region "Axis Setup"}
// Setup of Motion Commands for passthrough motor axis
MC_HomePassthrough(Axis := passthroughMotor);
MC_MovePassthrough(Axis := passthroughMotor);
MC_ResetPassthoughMotor(Axis := passthroughMotor);
MC_HaltPasstroughMotor(Axis := passthroughMotor);
{endregion}

{region "Timers"}
// If homing not complete within reasonable time, error out
homeTimeout(PT := homeTimeoutSetting);
// If passthrough doesn't reach setpoint in reasonable time, error out
movePassthroughTimeout();
{endregion}

{region "I/O and Fault Setup"}
// Passthrough position is based on reported motor position
actualPassthrough := passthroughMotor.ActPos;

// Setup simulation of I/O and faults for testing
simClose(in := cylinder.RetractAsserted, simFeedbackFault := UN00_Globals.simFaults.pressureBarFailedToMoveIn, inputToSimulate := PressureBarClosedSensor);
simOpen(in := cylinder.ExtendAsserted, simFeedbackFault := UN00_Globals.simFaults.pressureBarFailedToMoveOut, inputToSimulate := PressureBarOpenSensor);
ObstructionSensor.simulate := PressureBarClosedSensor.simulate := PressureBarOpenSensor.simulate := simulateIO;
ObstructionSensor.simValue := NOT UN00_Globals.simFaults.pressureBarObstucted;
EnableSimulation(device := cylinder, enableSim := simulateIO);

_isFullyClosed := PressureBarClosedSensor.Active;
_isFullyOpen := PressureBarOpenSensor.Active;

// Failed to reach sensor timers
// Exclusively use Close solonoid for Close fail timer since Open slow/low pressure uses both solenoids
failedToCloseTimer(IN := cylinder.RetractAsserted AND NOT _isFullyClosed,
					PT := faultTime,
					Q => failedToClose.faultTrigger);
failedToOpenTimer(IN := cylinder.ExtendAsserted AND NOT _isFullyOpen,
					PT := faultTime,
					Q => failedToOpen.faultTrigger);

// Obstruction fault is normally closed, fail safe.  Fault if collapsable jaw is broken anywhere outside of all the way in or all the way out
pressureBarObstructed.faultTrigger := ObstructionSensor.IsOff AND NOT (_isFullyClosed OR _isFullyOpen)
										OR ObstructionSensor.IsOff AND (_isFullyOpen AND cylinder.RetractAsserted);   // Also fault if broken when we try to close from all the way out
IF passthroughMotor.Error THEN
	motorFault.faultTrigger := TRUE;
	adjustablePassthroughState := 0;
ELSE
	motorFault.faultTrigger := FALSE;
END_IF
{endregion}

IF _reset THEN
	adjustablePassthroughState := 100;
	IF passthroughMotor.Error THEN
		MC_ResetPassthoughMotor.Execute := TRUE;
	END_IF
	_movePassthroughNow := FALSE;
	movePassthroughTimeout.IN := FALSE;
	_reset := FALSE;
END_IF

CASE adjustablePassthroughState OF

	0:  // Idle State.
		MC_ResetPassthoughMotor.Execute := FALSE;
		IF passthroughMotor.HomingDone
			AND NOT failedToClose.Active
			AND NOT failedToOpen.Active
			AND NOT failedToHome.Active
			AND NOT pressureBarObstructed.Active
			AND NOT motorFault.Active
			AND NOT failedToMovePassthrough.Active
			AND InDesiredPosition
		THEN
			_ready := TRUE;
		ELSE
			_ready := FALSE;
		END_IF

		IF _homeNow AND NOT passthroughMotor.HomingDone THEN
			MC_HomePassthrough.Execute := TRUE;
			OpenLowPressure();
			_homeNow := FALSE;
			adjustablePassthroughState := 1;
		ELSIF _homeNow AND passthroughMotor.HomingDone THEN
			_homeNow := FALSE;
		END_IF

		IF _movePassthroughNow AND passthroughMotor.HomingDone THEN
			IF InDesiredPosition THEN
				_movePassthroughNow := FALSE;
				adjustablePassthroughState := 100;
			ELSE
				MC_MovePassthrough.Position := passthroughSetting;
				MC_MovePassthrough.Velocity := ptVelo;
				MC_MovePassthrough.Acceleration := ptAccel;
				MC_MovePassthrough.Deceleration := ptDecel;
				_movePassthroughNow := FALSE;
				OpenLowPressure();

				IF UN00_Globals.simFaults.failedToMovePassthrough THEN
					movePassthroughTimeout.PT := TO_TIME(((ABS(actualPassthrough - passthroughSetting) / ptVelo) * 1000) - 500) ;
				ELSE
					movePassthroughTimeout.PT := TO_TIME(((ABS(actualPassthrough - passthroughSetting) / ptVelo) * 1000) + 2000);
				END_IF

				MC_MovePassthrough.Execute := TRUE;
				adjustablePassthroughState := 2;
			END_IF
		END_IF

	1:	// Homing
		homeTimeout.IN := TRUE;
		IF homeTimeout.Q
			OR MC_HomePassthrough.Error
			OR UN00_Globals.simFaults.pressureBarfailedToHome
		THEN
			failedToHome.Trigger();
			adjustablePassthroughState := 100;
		END_IF
		IF MC_HomePassthrough.Done THEN
			adjustablePassthroughState := 100;
		END_IF

	2:	// Start Moving Passthrough
		movePassthroughTimeout.IN := TRUE;

		IF MC_MovePassthrough.Error OR movePassthroughTimeout.Q THEN
			failedToMovePassthrough.Trigger();
			MC_MovePassthrough.Execute := FALSE;
			MC_HaltPasstroughMotor.Execute := TRUE;
			Exhaust();
			adjustablePassthroughState := 100;
		END_IF

		IF MC_MovePassthrough.Done THEN
			Open();
			MC_MovePassthrough.Execute := FALSE;
			adjustablePassthroughState := 100;
		END_IF

	100:// Cleanup
		MC_HomePassthrough.Execute := FALSE;
		//resetPassthoughMotor.Execute := FALSE;
		MC_MovePassthrough.Execute := FALSE;
		MC_HaltPasstroughMotor.Execute := FALSE;
		homeTimeout.IN := FALSE;
		movePassthroughTimeout.IN := FALSE;
		_homeNow := FALSE;

		adjustablePassthroughState := 0;

END_CASE

METHOD MovePassthrough
VAR_INPUT
	//passthroughSetting : REAL;
END_VAR

//_passthroughSetting := passthroughSetting;
_movePassthroughNow := TRUE;

{attribute 'monitoring' := 'variable'}
PROPERTY IsFullyOpen : BOOL

{attribute 'monitoring' := 'variable'}
PROPERTY IsFullyClosed : BOOL

METHOD Close

simClose.maxDelay := TO_DINT((actualPassthrough / 22.5) * 1000 + 50);
simClose.minDelay := TO_DINT((actualPassthrough / 22.5) * 1000 + 10);

cylinder.Retract();
faultTime := TO_TIME((actualPassthrough / 22.5) * 1000 + 300);

METHOD Open

simOpen.maxDelay := TO_INT((actualPassthrough / 22.5) * 1000 + 50);
simOpen.minDelay := TO_INT((actualPassthrough / 22.5) * 1000 + 10);

cylinder.Extend();
faultTime := TO_TIME((actualPassthrough / 22.5) * 1000 + 300);

METHOD RemovePower
VAR_INPUT
END_VAR

THIS^.Exhaust();
MC_HaltPasstroughMotor.Execute := TRUE;

PROPERTY IsHomed : BOOL

METHOD HomeNow
VAR_INPUT
END_VAR

_homeNow := TRUE;

METHOD OpenLowPressure
VAR_INPUT
END_VAR

simOpen.maxDelay := TO_INT((actualPassthrough / 4) * 1000 + 50);
simOpen.minDelay := TO_INT((actualPassthrough / 4) * 1000 + 10);
simOpen.faultDelay := simClose.maxDelay + 300;

ExtendLPIfPossible(cylinder);
faultTime := TO_TIME((actualPassthrough / 4) * 1000 + 300);

METHOD Exhaust
VAR_INPUT
END_VAR

ExhaustIfPossible(cylinder);

METHOD MoveNow
VAR_INPUT
END_VAR

THIS^.MovePassthrough();

PROPERTY InDesiredPosition : BOOL

(* ---- FB_Pro18BagDelivery.st ---- *)
FUNCTION_BLOCK FINAL FB_Pro18BagDelivery EXTENDS FB_BaseComponent IMPLEMENTS IBagDelivery
VAR_INPUT
	simulateIO : BOOL;
	printer : IPrinter;
	bagLength : REAL := 24.0;
	feedSpeed : REAL := 30.0;
	reverseSpeed : REAL := 3.0;
	printSpeed : REAL := 6.0;
	printOffset : REAL := 4.5;
	printLength : REAL := 6.0;
	maxReverseSetpoint : REAL := 3.0;
	sealOffset : REAL := 1.5;
	distanceFromSealBarToBagEdge : REAL := 3;
	distanceFromNipToBagEdge : REAL := 1.25;
	trapezoidalPercent : REAL := 0.1;
END_VAR
VAR_OUTPUT
	bagDeliveryFailedToMove : FB_Fault(name := Standard.CONCAT(_prefix,'Failed To Move'));
	bagFailedToSeparate : FB_Fault(name := Standard.CONCAT(_prefix,'Failed To Separate'));
END_VAR
VAR
	_feedAtPrintSpeed : BOOL;
	_feedBagOut : BOOL;
	_feedToPrintOffset : BOOL;
	_reverseToSeparate : BOOL;
	_bagFeedDone : BOOL;
	_bagSeparated : BOOL;
	_readyForPrint : BOOL;
	state : INT;
	nextState : INT;
	moveBagDeliveryTimeout : Standard.TON;
	MC_MoveBagDelivery : Sharp_Motion.MC_MoveRelative;
	MC_HaltBagDelivery : Sharp_Motion.MC_Halt;
	MC_ResetBagDelivery : Sharp_Motion.MC_Reset;
	remainingLength : REAL;
	bagReversedToPrintOffset : BOOL;
	bagEdgePhotoeyeSim : FB_SimulatedFeedbackPhysicalInput(name := 'Bag Edge Photoeye Sim');
END_VAR
VAR_IN_OUT
	bagDeliveryMotor : Sharp_Motion.Axis_REF;
	bagPhotoeyeInput : FB_PhysicalDigitalInput;
END_VAR
SUPER^();

{region "Axis Setup"}
// Setup of Motion Commands for Bag Delivery motor axis
MC_MoveBagDelivery(Axis := bagDeliveryMotor);
MC_HaltBagDelivery(Axis := bagDeliveryMotor);
MC_ResetBagDelivery(Axis := bagDeliveryMotor);
{endregion}
IF _reset THEN
	state := 100;
	nextState := 0;
	ClearStatus();
	IF bagDeliveryMotor.Error THEN
		MC_ResetBagDelivery.Execute := TRUE;
	END_IF
	_reset := FALSE;
END_IF

bagEdgePhotoeyeSim(
	in:= ,
	simFeedbackFault:= ,
	faultDelay:= ,
	minDelay:= 100,
	maxDelay:= 1000,
	Q=> ,
	fault=> ,
	inputToSimulate:= bagPhotoeyeInput);
//EnableSimulation(bagDeliveryMotor, simulateIO);
bagPhotoeyeInput.simulate := simulateIO;

IF trapezoidalPercent <= 0 THEN
	trapezoidalPercent := 0.1;
END_IF

CASE state OF
	0:		// Idle
			IF _feedBagOut THEN
				state := 10;
				_feedBagOut := FALSE;
				ClearStatus();
			END_IF

			IF _feedToPrintOffset THEN
				state := 20;
				_feedToPrintOffset := FALSE;
				ClearStatus();
			END_IF

			IF _reverseToSeparate THEN

				_bagSeparated := FALSE;
				state := 30;
				_reverseToSeparate := FALSE;
				ClearStatus();
			END_IF

			IF _feedAtPrintSpeed THEN
				state := 40;
				_feedAtPrintSpeed := FALSE;
				ClearStatus();
			END_IF

	1:		// Homing

	2:		//

	4: 		//

	5:		//

	6:		//

	7:		//

	10:		// Feed bag out
			MC_MoveBagDelivery.Acceleration := MC_MoveBagDelivery.Deceleration := (feedSpeed / trapezoidalPercent);
			MC_MoveBagDelivery.Velocity := feedSpeed;
			MC_MoveBagDelivery.Distance := remainingLength;
			moveBagDeliveryTimeout.PT := MoveTimeoutCalc(remainingLength, feedSpeed, 1000);
			moveBagDeliveryTimeout.IN := TRUE;
			MC_MoveBagDelivery.Execute := TRUE;
			_logger.AddLogItem(CONCAT(_prefix, 'Feeding Bag Out'));
			state := 101;
			nextState := 11;

	11:		// Set Bag Feed Done
			_bagFeedDone := TRUE;
			_logger.AddLogItem(CONCAT(_prefix, 'Bag Feed Done'));
			state := 0;
			nextState := 0;

	20:		// Feed bag to print offset.  If already at print offset from reversing, continue
			IF bagReversedToPrintOffset THEN
				state := 21;
				nextState := 0;
				bagReversedToPrintOffset := FALSE;
			ELSE
				MC_MoveBagDelivery.Acceleration := MC_MoveBagDelivery.Deceleration := (feedSpeed / trapezoidalPercent);
				MC_MoveBagDelivery.Velocity := feedSpeed;
				MC_MoveBagDelivery.Distance := printOffset;
				remainingLength := remainingLength - printOffset;
				moveBagDeliveryTimeout.PT := MoveTimeoutCalc(printOffset, feedSpeed, 1000);
				moveBagDeliveryTimeout.IN := TRUE;
				MC_MoveBagDelivery.Execute := TRUE;
				_logger.AddLogItem(CONCAT(_prefix, 'Feeding Bag to Print Offset'));
				state := 101;
				nextState := 21;
			END_IF

	21: 	// Set Ready For Print
			_readyForPrint := TRUE;
			state := 0;
			nextState := 0;

	30:		// Reverse to Separate
			MC_MoveBagDelivery.Acceleration := MC_MoveBagDelivery.Deceleration := (reverseSpeed / trapezoidalPercent);
			MC_MoveBagDelivery.Velocity := reverseSpeed;
			MC_MoveBagDelivery.Distance := maxReverseSetpoint;
			moveBagDeliveryTimeout.PT := MoveTimeoutCalc(maxReverseSetpoint, reverseSpeed, 1000);
			moveBagDeliveryTimeout.IN := TRUE;
			MC_MoveBagDelivery.Execute := TRUE;
			_logger.AddLogItem(CONCAT(_prefix, 'Reversing to Photoeye'));
			bagEdgePhotoeyeSim.in := TRUE;
			state := 31;
			//nextState := 31;

	31:		// Stop bag once edge clears photoeye. If move command finishes that means the bag didn't separate
			IF MC_MoveBagDelivery.Done THEN
				bagFailedToSeparate.Trigger();
				ClearStatus();
				state := 100;
				nextState := 0;
			END_IF

			IF MC_MoveBagDelivery.Error OR moveBagDeliveryTimeout.Q THEN
				bagDeliveryFailedToMove.Trigger();
				MC_MoveBagDelivery.Execute := FALSE;
				MC_HaltBagDelivery.Execute := TRUE;
				ClearStatus();
				nextState := 0;
				state := 100;
			END_IF

			IF bagPhotoeyeInput.Active THEN
				MC_MoveBagDelivery.Execute := FALSE;
				MC_HaltBagDelivery.Execute := TRUE;
				bagEdgePhotoeyeSim.in := FALSE;
				state := 32;
			END_IF

	32: 	// Set Bag Reversed OR reverse further for zero print datum if needed
			IF MC_HaltBagDelivery.Done THEN
				MC_HaltBagDelivery.Execute := FALSE;
				IF NOT printer.OptionActive OR
				   printOffset >= distanceFromNipToBagEdge
				THEN
					remainingLength := bagLength + printOffset;
					_bagSeparated := TRUE;
					state := 0;
					nextState := 0;
				ELSE
					state := 33;
				END_IF
			END_IF

	33: 	// Reverse to Nip for zero print datum
			MC_MoveBagDelivery.Acceleration := MC_MoveBagDelivery.Deceleration := (reverseSpeed / trapezoidalPercent);
			MC_MoveBagDelivery.Velocity := reverseSpeed;
			MC_MoveBagDelivery.Distance := (distanceFromNipToBagEdge - printOffset) * -1;
			moveBagDeliveryTimeout.PT := MoveTimeoutCalc(distanceFromNipToBagEdge, reverseSpeed, 1000);
			moveBagDeliveryTimeout.IN := TRUE;
			MC_MoveBagDelivery.Execute := TRUE;
			_logger.AddLogItem(CONCAT(_prefix, 'Reversing to Nip'));
			remainingLength := remainingLength + distanceFromNipToBagEdge;
			state := 101;
			nextState := 34;

	34: 	_bagSeparated := TRUE;
			//_readyForPrint := TRUE;
			state := 0;
			nextState := 0;

	40:		// Feed at Print Speed
			MC_MoveBagDelivery.Acceleration := MC_MoveBagDelivery.Deceleration := (reverseSpeed / trapezoidalPercent);
			MC_MoveBagDelivery.Velocity := reverseSpeed;
			MC_MoveBagDelivery.Distance := printLength;
			moveBagDeliveryTimeout.PT := MoveTimeoutCalc(distanceFromNipToBagEdge, reverseSpeed, 1000);
			moveBagDeliveryTimeout.IN := TRUE;
			MC_MoveBagDelivery.Execute := TRUE;
			_logger.AddLogItem(CONCAT(_prefix, 'Feeding At Print Speed'));
			remainingLength := remainingLength - printLength;
			state := 101;
			nextState := 0;

	100:	// Cleanup
			MC_MoveBagDelivery.Execute := FALSE;
			MC_HaltBagDelivery.Execute := FALSE;
			moveBagDeliveryTimeout.IN := FALSE;
			bagEdgePhotoeyeSim.in := FALSE;
			state := nextState;

	101: 	// Wait for Move to complete
			IF MC_MoveBagDelivery.Error OR moveBagDeliveryTimeout.Q THEN
				bagDeliveryFailedToMove.Trigger();
				MC_MoveBagDelivery.Execute := FALSE;
				MC_HaltBagDelivery.Execute := TRUE;
				ClearStatus();
				nextState := 0;
				state := 100;
			END_IF

			IF MC_MoveBagDelivery.Done THEN
				moveBagDeliveryTimeout.IN := FALSE;
				MC_MoveBagDelivery.Execute := FALSE;
				state := nextState;
			END_IF

	103:	// Set In Position and go back to idle

			nextState := 0;
			state := 100;

END_CASE

METHOD FeedToPhotoeye
VAR_INPUT
END_VAR

{attribute 'monitoring' := 'variable'}
PROPERTY BagFeedDone : BOOL

{attribute 'monitoring' := 'variable'}
PROPERTY BagSeparated : BOOL

{attribute 'monitoring' := 'variable'}
PROPERTY ReadyForPrint : BOOL

METHOD ReverseToSeparate

_reverseToSeparate := TRUE;

METHOD FeedToPrintOffset

_feedToPrintOffset := TRUE;

METHOD FeedAtPrintSpeed

_feedAtPrintSpeed := TRUE;

METHOD FeedBagOut

_feedBagOut := TRUE;

METHOD ClearStatus
VAR_INPUT
END_VAR

_bagFeedDone := FALSE;
_bagSeparated := FALSE;
_readyForPrint := FALSE;

FUNCTION_BLOCK FINAL FB_Pro18BagDelivery EXTENDS FB_BaseComponent IMPLEMENTS IBagDelivery
VAR_INPUT
	simulateIO : BOOL;
	printer : IPrinter;
	bagLength : REAL := 24.0;
	feedSpeed : REAL := 30.0;
	reverseSpeed : REAL := 3.0;
	printSpeed : REAL := 6.0;
	printOffset : REAL := 4.5;
	printLength : REAL := 6.0;
	maxReverseSetpoint : REAL := 3.0;
	sealOffset : REAL := 1.5;
	distanceFromSealBarToBagEdge : REAL := 3;
	distanceFromNipToBagEdge : REAL := 1.25;
	trapezoidalPercent : REAL := 0.1;
END_VAR
VAR_OUTPUT
	bagDeliveryFailedToMove : FB_Fault(name := Standard.CONCAT(_prefix,'Failed To Move'));
	bagFailedToSeparate : FB_Fault(name := Standard.CONCAT(_prefix,'Failed To Separate'));
END_VAR
VAR
	_feedAtPrintSpeed : BOOL;
	_feedBagOut : BOOL;
	_feedToPrintOffset : BOOL;
	_reverseToSeparate : BOOL;
	_bagFeedDone : BOOL;
	_bagSeparated : BOOL;
	_readyForPrint : BOOL;
	state : INT;
	nextState : INT;
	moveBagDeliveryTimeout : Standard.TON;
	MC_MoveBagDelivery : Sharp_Motion.MC_MoveRelative;
	MC_HaltBagDelivery : Sharp_Motion.MC_Halt;
	MC_ResetBagDelivery : Sharp_Motion.MC_Reset;
	remainingLength : REAL;
	bagReversedToPrintOffset : BOOL;
	bagEdgePhotoeyeSim : FB_SimulatedFeedbackPhysicalInput(name := 'Bag Edge Photoeye Sim');
END_VAR
VAR_IN_OUT
	bagDeliveryMotor : Sharp_Motion.Axis_REF;
	bagPhotoeyeInput : FB_PhysicalDigitalInput;
END_VAR
SUPER^();

{region "Axis Setup"}
// Setup of Motion Commands for Bag Delivery motor axis
MC_MoveBagDelivery(Axis := bagDeliveryMotor);
MC_HaltBagDelivery(Axis := bagDeliveryMotor);
MC_ResetBagDelivery(Axis := bagDeliveryMotor);
{endregion}
IF _reset THEN
	state := 100;
	nextState := 0;
	ClearStatus();
	IF bagDeliveryMotor.Error THEN
		MC_ResetBagDelivery.Execute := TRUE;
	END_IF
	_reset := FALSE;
END_IF

bagEdgePhotoeyeSim(
	in:= ,
	simFeedbackFault:= ,
	faultDelay:= ,
	minDelay:= 100,
	maxDelay:= 1000,
	Q=> ,
	fault=> ,
	inputToSimulate:= bagPhotoeyeInput);
//EnableSimulation(bagDeliveryMotor, simulateIO);
bagPhotoeyeInput.simulate := simulateIO;

IF trapezoidalPercent <= 0 THEN
	trapezoidalPercent := 0.1;
END_IF

CASE state OF
	0:		// Idle
			IF _feedBagOut THEN
				state := 10;
				_feedBagOut := FALSE;
				ClearStatus();
			END_IF

			IF _feedToPrintOffset THEN
				state := 20;
				_feedToPrintOffset := FALSE;
				ClearStatus();
			END_IF

			IF _reverseToSeparate THEN

				_bagSeparated := FALSE;
				state := 30;
				_reverseToSeparate := FALSE;
				ClearStatus();
			END_IF

			IF _feedAtPrintSpeed THEN
				state := 40;
				_feedAtPrintSpeed := FALSE;
				ClearStatus();
			END_IF

	1:		// Homing

	2:		//

	4: 		//

	5:		//

	6:		//

	7:		//

	10:		// Feed bag out
			MC_MoveBagDelivery.Acceleration := MC_MoveBagDelivery.Deceleration := (feedSpeed / trapezoidalPercent);
			MC_MoveBagDelivery.Velocity := feedSpeed;
			MC_MoveBagDelivery.Distance := remainingLength;
			moveBagDeliveryTimeout.PT := MoveTimeoutCalc(remainingLength, feedSpeed, 1000);
			moveBagDeliveryTimeout.IN := TRUE;
			MC_MoveBagDelivery.Execute := TRUE;
			_logger.AddLogItem(CONCAT(_prefix, 'Feeding Bag Out'));
			state := 101;
			nextState := 11;

	11:		// Set Bag Feed Done
			_bagFeedDone := TRUE;
			_logger.AddLogItem(CONCAT(_prefix, 'Bag Feed Done'));
			state := 0;
			nextState := 0;

	20:		// Feed bag to print offset.  If already at print offset from reversing, continue
			IF bagReversedToPrintOffset THEN
				state := 21;
				nextState := 0;
				bagReversedToPrintOffset := FALSE;
			ELSE
				MC_MoveBagDelivery.Acceleration := MC_MoveBagDelivery.Deceleration := (feedSpeed / trapezoidalPercent);
				MC_MoveBagDelivery.Velocity := feedSpeed;
				MC_MoveBagDelivery.Distance := printOffset;
				remainingLength := remainingLength - printOffset;
				moveBagDeliveryTimeout.PT := MoveTimeoutCalc(printOffset, feedSpeed, 1000);
				moveBagDeliveryTimeout.IN := TRUE;
				MC_MoveBagDelivery.Execute := TRUE;
				_logger.AddLogItem(CONCAT(_prefix, 'Feeding Bag to Print Offset'));
				state := 101;
				nextState := 21;
			END_IF

	21: 	// Set Ready For Print
			_readyForPrint := TRUE;
			state := 0;
			nextState := 0;

	30:		// Reverse to Separate
			MC_MoveBagDelivery.Acceleration := MC_MoveBagDelivery.Deceleration := (reverseSpeed / trapezoidalPercent);
			MC_MoveBagDelivery.Velocity := reverseSpeed;
			MC_MoveBagDelivery.Distance := maxReverseSetpoint;
			moveBagDeliveryTimeout.PT := MoveTimeoutCalc(maxReverseSetpoint, reverseSpeed, 1000);
			moveBagDeliveryTimeout.IN := TRUE;
			MC_MoveBagDelivery.Execute := TRUE;
			_logger.AddLogItem(CONCAT(_prefix, 'Reversing to Photoeye'));
			bagEdgePhotoeyeSim.in := TRUE;
			state := 31;
			//nextState := 31;

	31:		// Stop bag once edge clears photoeye. If move command finishes that means the bag didn't separate
			IF MC_MoveBagDelivery.Done THEN
				bagFailedToSeparate.Trigger();
				ClearStatus();
				state := 100;
				nextState := 0;
			END_IF

			IF MC_MoveBagDelivery.Error OR moveBagDeliveryTimeout.Q THEN
				bagDeliveryFailedToMove.Trigger();
				MC_MoveBagDelivery.Execute := FALSE;
				MC_HaltBagDelivery.Execute := TRUE;
				ClearStatus();
				nextState := 0;
				state := 100;
			END_IF

			IF bagPhotoeyeInput.Active THEN
				MC_MoveBagDelivery.Execute := FALSE;
				MC_HaltBagDelivery.Execute := TRUE;
				bagEdgePhotoeyeSim.in := FALSE;
				state := 32;
			END_IF

	32: 	// Set Bag Reversed OR reverse further for zero print datum if needed
			IF MC_HaltBagDelivery.Done THEN
				MC_HaltBagDelivery.Execute := FALSE;
				IF NOT printer.OptionActive OR
				   printOffset >= distanceFromNipToBagEdge
				THEN
					remainingLength := bagLength + printOffset;
					_bagSeparated := TRUE;
					state := 0;
					nextState := 0;
				ELSE
					state := 33;
				END_IF
			END_IF

	33: 	// Reverse to Nip for zero print datum
			MC_MoveBagDelivery.Acceleration := MC_MoveBagDelivery.Deceleration := (reverseSpeed / trapezoidalPercent);
			MC_MoveBagDelivery.Velocity := reverseSpeed;
			MC_MoveBagDelivery.Distance := (distanceFromNipToBagEdge - printOffset) * -1;
			moveBagDeliveryTimeout.PT := MoveTimeoutCalc(distanceFromNipToBagEdge, reverseSpeed, 1000);
			moveBagDeliveryTimeout.IN := TRUE;
			MC_MoveBagDelivery.Execute := TRUE;
			_logger.AddLogItem(CONCAT(_prefix, 'Reversing to Nip'));
			remainingLength := remainingLength + distanceFromNipToBagEdge;
			state := 101;
			nextState := 34;

	34: 	_bagSeparated := TRUE;
			//_readyForPrint := TRUE;
			state := 0;
			nextState := 0;

	40:		// Feed at Print Speed
			MC_MoveBagDelivery.Acceleration := MC_MoveBagDelivery.Deceleration := (reverseSpeed / trapezoidalPercent);
			MC_MoveBagDelivery.Velocity := reverseSpeed;
			MC_MoveBagDelivery.Distance := printLength;
			moveBagDeliveryTimeout.PT := MoveTimeoutCalc(distanceFromNipToBagEdge, reverseSpeed, 1000);
			moveBagDeliveryTimeout.IN := TRUE;
			MC_MoveBagDelivery.Execute := TRUE;
			_logger.AddLogItem(CONCAT(_prefix, 'Feeding At Print Speed'));
			remainingLength := remainingLength - printLength;
			state := 101;
			nextState := 0;

	100:	// Cleanup
			MC_MoveBagDelivery.Execute := FALSE;
			MC_HaltBagDelivery.Execute := FALSE;
			moveBagDeliveryTimeout.IN := FALSE;
			bagEdgePhotoeyeSim.in := FALSE;
			state := nextState;

	101: 	// Wait for Move to complete
			IF MC_MoveBagDelivery.Error OR moveBagDeliveryTimeout.Q THEN
				bagDeliveryFailedToMove.Trigger();
				MC_MoveBagDelivery.Execute := FALSE;
				MC_HaltBagDelivery.Execute := TRUE;
				ClearStatus();
				nextState := 0;
				state := 100;
			END_IF

			IF MC_MoveBagDelivery.Done THEN
				moveBagDeliveryTimeout.IN := FALSE;
				MC_MoveBagDelivery.Execute := FALSE;
				state := nextState;
			END_IF

	103:	// Set In Position and go back to idle

			nextState := 0;
			state := 100;

END_CASE

METHOD FeedToPhotoeye
VAR_INPUT
END_VAR

{attribute 'monitoring' := 'variable'}
PROPERTY BagFeedDone : BOOL

{attribute 'monitoring' := 'variable'}
PROPERTY BagSeparated : BOOL

{attribute 'monitoring' := 'variable'}
PROPERTY ReadyForPrint : BOOL

METHOD ReverseToSeparate

_reverseToSeparate := TRUE;

METHOD FeedToPrintOffset

_feedToPrintOffset := TRUE;

METHOD FeedAtPrintSpeed

_feedAtPrintSpeed := TRUE;

METHOD FeedBagOut

_feedBagOut := TRUE;

METHOD ClearStatus
VAR_INPUT
END_VAR

_bagFeedDone := FALSE;
_bagSeparated := FALSE;
_readyForPrint := FALSE;

(* ---- FB_Pro18ZebraPrinter.st ---- *)
FUNCTION_BLOCK FINAL FB_Pro18ZebraPrinter EXTENDS FB_BasicPrinter
VAR_INPUT
	printHead : IUpDown;
	printHeadDebounceSetpoint : TIME;
END_VAR
VAR_OUTPUT
	serviceRequired : FB_Fault(name := Standard.CONCAT(_prefix,'Service Required'));
	ribbonLow : Warning;
END_VAR
VAR
	printHeadDebounceTimer : Standard.TON;
	printerPrintingONS : FB_ONS;
	printDoneSim : FB_MonostableMultivibrator(name := 'Print Done Sim=');
END_VAR
VAR_IN_OUT
	dataReadyInput : FB_PhysicalDigitalInput;
	serviceRequiredInput : FB_PhysicalDigitalInput;
	ribbonLowInput : FB_PhysicalDigitalInput;
	endOfPrintInput : FB_PhysicalDigitalInput;
	startPrintOutput : FB_PhysicalDigitalOutput;
	ribbonUnwindRunOutput : FB_PhysicalDigitalOutput;
END_VAR

//	Function Block: FB_Pro18ZebraPrinter()
//	Description: Pro-18 Zebra Printer
//				 Printer applicator should be in Mode 2, in which the End Of Print input stays high while printing,
//				 this way we can release the print head and not waste ribbon if the label is shorter than
//	Created by: Ben Hess
//	Created Date: Thursday, August 1st, 2019

SUPER^();

// Setup of inputs and faults, warnings
_hasLabel := dataReadyInput.Active OR simulateIO;

IF serviceRequiredInput.Active AND THIS^.OptionEnabled THEN
	serviceRequired.Trigger();
END_IF

ribbonLow.active := ribbonLowInput.Active AND THIS^.OptionEnabled;

// Simulation setup
EnableSimulation(printHead, simulateIO);
EnableSimulation(startPrintOutput, simulateIO);
EnableSimulation(ribbonUnwindRunOutput, simulateIO);
endOfPrintInput.simulate := simulateIO;
endOfPrintInput.simValue := printDoneSim.Q;

printDoneSim.DwellSetting := TO_UINT(((printLength / TO_REAL(printSpeed)) * 1000) + 50.0);
printDoneSim();

printHeadDebounceTimer(PT := printHeadDebounceSetpoint);
printerPrintingONS(CLK := endOfPrintInput.Active);

IF _reset THEN
	state := 100;
	_reset := FALSE;
END_IF

CASE state OF
	0:		// Idle
			IF _beginPrinting AND THIS^.OptionEnabled THEN
				state := 10;
				_printDone := FALSE;
				_beginPrinting := FALSE;
			END_IF

	10:		// Start Print cycle
			printHead.MoveDown();
			printHeadDebounceTimer.IN := TRUE;
			_logger.AddLogItem(CONCAT(_prefix, 'Print Started'));
			state := 11;

	11:		//Wait for print head debounce
			IF printHeadDebounceTimer.Q THEN
				printHeadDebounceTimer.IN := FALSE;
				startPrintOutput.TurnOn();
				ribbonUnwindRunOutput.TurnOn();
				printDoneSim.Trigger();
				state := 12;
				_printing := TRUE;
			END_IF

	12:		// Print until finished or faulted
			IF printerPrintingONS.OSF OR serviceRequired.FaultActive THEN
				startPrintOutput.TurnOff();
				ribbonUnwindRunOutput.TurnOff();
				printHead.MoveUp();
				_printing := FALSE;
				_printDone := TRUE;
				_logger.AddLogItem(CONCAT(_prefix, 'Print Done'));
				state := 0;
			END_IF

	100:	// Clear status
			_printing := FALSE;
			_beginPrinting := FALSE;
			_printDone := FALSE;
			printDoneSim.ManualOff();
			startPrintOutput.TurnOff();
			ribbonUnwindRunOutput.TurnOff();
			printHeadDebounceTimer.IN := FALSE;
			state := 0;
END_CASE

(* ---- FB_SimBasicBagDelivery.st ---- *)
FUNCTION_BLOCK FB_SimBasicBagDelivery EXTENDS FB_BaseComponent IMPLEMENTS IBagDelivery, IExecuteAutomatically
VAR_INPUT
	feedSpeed : UDINT;
	reverseSpeed : UDINT;
	printSpeed : UDINT;
	printLength : REAL;
	bagLength : REAL;
	reverseLength : REAL;
	printOffset : REAL;
END_VAR
VAR_OUTPUT
END_VAR

VAR
	feedAtPrintSpeed : FB_SimulatedFeedback(name := CONCAT(_prefix,'Feed at Print Speed'));
	feedBagOut : FB_SimulatedFeedback(name := CONCAT(_prefix,'Feed Bag Out'));
	feedToPrintOffset : FB_SimulatedFeedback(name := CONCAT(_prefix,'Feed to Print Offset'));
	reverseToSeparate : FB_SimulatedFeedback(name := CONCAT(_prefix,'Reverse to Separate'));
END_VAR

{attribute 'monitoring' := 'variable'}
PROPERTY BagFeedDone : BOOL

METHOD PRIVATE ClearStatus
VAR_INPUT
END_VAR

feedAtPrintSpeed.in := FALSE;
feedBagOut.in := FALSE;
feedToPrintOffset.in := FALSE;
reverseToSeparate.in := FALSE;
THIS^.Execute();

{attribute 'monitoring' := 'variable'}
PROPERTY BagSeparated : BOOL

{attribute 'monitoring' := 'variable'}
PROPERTY ReadyForPrint : BOOL

METHOD ReverseToSeparate

ClearStatus();
reverseToSeparate.maxDelay := TO_DINT(((reverseLength / TO_REAL(reverseSpeed)) * 1000) + 50.0);
reverseToSeparate.minDelay := TO_DINT(((reverseLength / TO_REAL(reverseSpeed)) * 1000) + 10.0);
reverseToSeparate.in := TRUE;

METHOD FeedToPrintOffset

ClearStatus();
feedToPrintOffset.maxDelay := TO_DINT(((printOffset / TO_REAL(feedSpeed)) * 1000) + 50.0);
feedToPrintOffset.minDelay := TO_DINT(((printOffset / TO_REAL(feedSpeed)) * 1000) + 20.0);
feedToPrintOffset.in := TRUE;

METHOD FeedAtPrintSpeed

ClearStatus();
feedAtPrintSpeed.maxDelay := TO_DINT(((printLength / TO_REAL(printSpeed)) * 1000) + 50.0);
feedAtPrintSpeed.minDelay := TO_DINT(((printLength / TO_REAL(printSpeed)) * 1000) + 10.0);
feedAtPrintSpeed.in := TRUE;

METHOD FeedBagOut

ClearStatus();
feedBagOut.maxDelay := TO_DINT(((bagLength / TO_REAL(feedSpeed)) * 1000) + 50.0);
feedBagOut.minDelay := TO_DINT(((bagLength / TO_REAL(feedSpeed)) * 1000) + 10.0);
feedBagOut.in := TRUE;

METHOD Execute

SUPER^.Execute();
feedAtPrintSpeed();
feedBagOut();
feedToPrintOffset();
reverseToSeparate();

METHOD FeedToPhotoeye
VAR_INPUT
END_VAR

FUNCTION_BLOCK FB_SimBasicBagDelivery EXTENDS FB_BaseComponent IMPLEMENTS IBagDelivery, IExecuteAutomatically
VAR_INPUT
	feedSpeed : UDINT;
	reverseSpeed : UDINT;
	printSpeed : UDINT;
	printLength : REAL;
	bagLength : REAL;
	reverseLength : REAL;
	printOffset : REAL;
END_VAR
VAR_OUTPUT
END_VAR

VAR
	feedAtPrintSpeed : FB_SimulatedFeedback(name := CONCAT(_prefix,'Feed at Print Speed'));
	feedBagOut : FB_SimulatedFeedback(name := CONCAT(_prefix,'Feed Bag Out'));
	feedToPrintOffset : FB_SimulatedFeedback(name := CONCAT(_prefix,'Feed to Print Offset'));
	reverseToSeparate : FB_SimulatedFeedback(name := CONCAT(_prefix,'Reverse to Separate'));
END_VAR

{attribute 'monitoring' := 'variable'}
PROPERTY BagFeedDone : BOOL

METHOD PRIVATE ClearStatus
VAR_INPUT
END_VAR

feedAtPrintSpeed.in := FALSE;
feedBagOut.in := FALSE;
feedToPrintOffset.in := FALSE;
reverseToSeparate.in := FALSE;
THIS^.Execute();

{attribute 'monitoring' := 'variable'}
PROPERTY BagSeparated : BOOL

{attribute 'monitoring' := 'variable'}
PROPERTY ReadyForPrint : BOOL

METHOD ReverseToSeparate

ClearStatus();
reverseToSeparate.maxDelay := TO_DINT(((reverseLength / TO_REAL(reverseSpeed)) * 1000) + 50.0);
reverseToSeparate.minDelay := TO_DINT(((reverseLength / TO_REAL(reverseSpeed)) * 1000) + 10.0);
reverseToSeparate.in := TRUE;

METHOD FeedToPrintOffset

ClearStatus();
feedToPrintOffset.maxDelay := TO_DINT(((printOffset / TO_REAL(feedSpeed)) * 1000) + 50.0);
feedToPrintOffset.minDelay := TO_DINT(((printOffset / TO_REAL(feedSpeed)) * 1000) + 20.0);
feedToPrintOffset.in := TRUE;

METHOD FeedAtPrintSpeed

ClearStatus();
feedAtPrintSpeed.maxDelay := TO_DINT(((printLength / TO_REAL(printSpeed)) * 1000) + 50.0);
feedAtPrintSpeed.minDelay := TO_DINT(((printLength / TO_REAL(printSpeed)) * 1000) + 10.0);
feedAtPrintSpeed.in := TRUE;

METHOD FeedBagOut

ClearStatus();
feedBagOut.maxDelay := TO_DINT(((bagLength / TO_REAL(feedSpeed)) * 1000) + 50.0);
feedBagOut.minDelay := TO_DINT(((bagLength / TO_REAL(feedSpeed)) * 1000) + 10.0);
feedBagOut.in := TRUE;

METHOD Execute

SUPER^.Execute();
feedAtPrintSpeed();
feedBagOut();
feedToPrintOffset();
reverseToSeparate();

METHOD FeedToPhotoeye
VAR_INPUT
END_VAR

(* ---- FB_SimBasicExitConveyor.st ---- *)
FUNCTION_BLOCK FB_SimBasicExitConveyor EXTENDS FB_BaseComponent IMPLEMENTS IExitConveyor, IExecuteAutomatically
VAR_INPUT
END_VAR
VAR_OUTPUT
END_VAR
VAR
END_VAR

METHOD BeginDischarge

_logger.AddLogItem(CONCAT(_prefix, 'Begin Discharge'));

FUNCTION_BLOCK FB_SimBasicExitConveyor EXTENDS FB_BaseComponent IMPLEMENTS IExitConveyor, IExecuteAutomatically
VAR_INPUT
END_VAR
VAR_OUTPUT
END_VAR
VAR
END_VAR

METHOD BeginDischarge

_logger.AddLogItem(CONCAT(_prefix, 'Begin Discharge'));

(* ---- FB_SimBasicLoadPlate.st ---- *)
FUNCTION_BLOCK FB_SimBasicLoadPlate EXTENDS FB_BaseComponent IMPLEMENTS IRetractingLoadPlate, IExecuteAutomatically
VAR_INPUT
	loadPlateDwell : REAL := 2.5;
END_VAR
VAR_OUTPUT
END_VAR
VAR
	beginDischarge : FB_SimulatedFeedback(name := CONCAT(_prefix,'Begin Discharge'));
END_VAR

PROPERTY ReadyToLoad : BOOL

METHOD Execute

SUPER^.Execute();
beginDischarge();

METHOD BeginDischarge

ClearStatus();
beginDischarge.maxDelay := TO_INT(loadPlateDwell * 1000.0 + 600.0);
beginDischarge.minDelay := TO_INT(loadPlateDwell * 1000.0 + 400.0);
beginDischarge.in := TRUE;

METHOD PRIVATE ClearStatus
VAR_INPUT
END_VAR

beginDischarge.in := FALSE;
THIS^.Execute();

(* ---- FB_SimBasicPrinter.st ---- *)
FUNCTION_BLOCK FB_SimBasicPrinter EXTENDS FB_BaseComponent IMPLEMENTS IPrinter, IExecuteAutomatically
VAR_INPUT
	printSpeed : UDINT;
	printLength : REAL;
END_VAR
VAR_OUTPUT
END_VAR
VAR
	beginPrinting : FB_SimulatedFeedback(name := CONCAT(_prefix,'Begin Printing'));
END_VAR

{attribute 'monitoring' := 'variable'}
PROPERTY HasLabel : BOOL

METHOD ClearStatus : BOOL
VAR_INPUT
END_VAR

beginPrinting.in := FALSE;
THIS^.Execute();

{attribute 'monitoring' := 'variable'}
PROPERTY PrintDone : BOOL

METHOD BeginPrinting

ClearStatus();
beginPrinting.maxDelay := TO_DINT(((printLength / TO_REAL(printSpeed)) * 1000) + 50.0);
beginPrinting.minDelay := TO_DINT(((printLength / TO_REAL(printSpeed)) * 1000) + 10.0);
beginPrinting.in := TRUE;

METHOD Execute

SUPER^.Execute();
beginPrinting();

FUNCTION_BLOCK FB_SimBasicPrinter EXTENDS FB_BaseComponent IMPLEMENTS IPrinter, IExecuteAutomatically
VAR_INPUT
	printSpeed : UDINT;
	printLength : REAL;
END_VAR
VAR_OUTPUT
END_VAR
VAR
	beginPrinting : FB_SimulatedFeedback(name := CONCAT(_prefix,'Begin Printing'));
END_VAR

{attribute 'monitoring' := 'variable'}
PROPERTY HasLabel : BOOL

METHOD ClearStatus : BOOL
VAR_INPUT
END_VAR

beginPrinting.in := FALSE;
THIS^.Execute();

{attribute 'monitoring' := 'variable'}
PROPERTY PrintDone : BOOL

METHOD BeginPrinting

ClearStatus();
beginPrinting.maxDelay := TO_DINT(((printLength / TO_REAL(printSpeed)) * 1000) + 50.0);
beginPrinting.minDelay := TO_DINT(((printLength / TO_REAL(printSpeed)) * 1000) + 10.0);
beginPrinting.in := TRUE;

METHOD Execute

SUPER^.Execute();
beginPrinting();

(* ---- FB_SimBasicSealFlatteners.st ---- *)
FUNCTION_BLOCK FB_SimBasicSealFlatteners EXTENDS FB_BaseComponent IMPLEMENTS ISealFlatteners, IExecuteAutomatically
VAR_INPUT
END_VAR
VAR_OUTPUT
END_VAR
VAR
	_inPosition : BOOL;
	moveToBagFeed : FB_SimulatedFeedback(name := CONCAT(_prefix,'Move to Bag Feed')) := (minDelay := 20, maxDelay := 100);
	moveToBagHolding : FB_SimulatedFeedback(name := CONCAT(_prefix,'Move to Bag Holding')) := (minDelay := 190, maxDelay := 210);
	moveToClearance : FB_SimulatedFeedback(name := CONCAT(_prefix,'Move to Clearance')) := (minDelay := 50, maxDelay := 70);
	moveToSeal : FB_SimulatedFeedback(name := CONCAT(_prefix,'Move to Sealing')) := (minDelay := 200, maxDelay := 250);
	moveToIn : FB_SimulatedFeedback(name := CONCAT(_prefix,'Move to In')) := (minDelay := 200, maxDelay := 250);
	okayToMove : BOOL;
END_VAR

{attribute 'monitoring' := 'variable'}
PROPERTY InPosition : BOOL

METHOD ToSeal

ClearStatus();
moveToSeal.in := TRUE;

METHOD ToClearance

ClearStatus();
moveToClearance.in := TRUE;

METHOD ToBagFeed

ClearStatus();
moveToBagFeed.in := TRUE;

METHOD ToIn

ClearStatus();
moveToIn.in := TRUE;

METHOD BagIsOpen

ClearStatus();
moveToBagHolding.in := TRUE;

METHOD Execute

SUPER^.Execute();
moveToBagFeed();
moveToBagHolding();
moveToClearance();
moveToSeal();
moveToIn();

METHOD PRIVATE ClearStatus
VAR_INPUT
END_VAR

moveToBagFeed.in := FALSE;
moveToBagHolding.in := FALSE;
moveToClearance.in := FALSE;
moveToSeal.in := FALSE;
moveToIn.in := FALSE;
THIS^.Execute();

(* ---- FB_SimBasicVacuum.st ---- *)
FUNCTION_BLOCK FB_SimBasicVacuum EXTENDS FB_BaseComponent IMPLEMENTS IVacuumBagOpen, IExecuteAutomatically
VAR_INPUT
	vacGrabDwell : REAL;
END_VAR
VAR_OUTPUT
END_VAR
VAR
	startVac : FB_SimulatedFeedback(name := CONCAT(_prefix,'Start Vac'));
END_VAR

{attribute 'monitoring' := 'variable'}
PROPERTY VacuumOn : BOOL

METHOD PRIVATE ClearStatus
VAR_INPUT
END_VAR

startVac.in := FALSE;
THIS^.Execute();

METHOD StartVacuum

ClearStatus();
startVac.maxDelay := TO_INT(vacGrabDwell * 1000.0 + 10.0);
startVac.minDelay := TO_INT(vacGrabDwell * 1000.0 - 10.0);
startVac.in := TRUE;

METHOD StopVacuum

startVac.in := FALSE;
THIS^.Execute();

METHOD Execute

SUPER^.Execute();
startVac();

FUNCTION_BLOCK FB_SimBasicVacuum EXTENDS FB_BaseComponent IMPLEMENTS IVacuumBagOpen, IExecuteAutomatically
VAR_INPUT
	vacGrabDwell : REAL;
END_VAR
VAR_OUTPUT
END_VAR
VAR
	startVac : FB_SimulatedFeedback(name := CONCAT(_prefix,'Start Vac'));
END_VAR

{attribute 'monitoring' := 'variable'}
PROPERTY VacuumOn : BOOL

METHOD PRIVATE ClearStatus
VAR_INPUT
END_VAR

startVac.in := FALSE;
THIS^.Execute();

METHOD StartVacuum

ClearStatus();
startVac.maxDelay := TO_INT(vacGrabDwell * 1000.0 + 10.0);
startVac.minDelay := TO_INT(vacGrabDwell * 1000.0 - 10.0);
startVac.in := TRUE;

METHOD StopVacuum

startVac.in := FALSE;
THIS^.Execute();

METHOD Execute

SUPER^.Execute();
startVac();

(* ---- FB_SimMotor.st ---- *)
FUNCTION_BLOCK FB_SimMotor EXTENDS Sharp_Motion.Axis_REF
VAR_INPUT
	simFault : BOOL;
END_VAR
VAR_OUTPUT
END_VAR
VAR
	homingTimer : Standard.TON;
	movingTimer : Standard.TON;
	resetTimer : Standard.TON := (PT := T#500ms);
	state : INT;
	homingState : INT;
	moveAbsState : INT;
	moveRelState : INT;
	_reset : BOOL;
	distanceToMove : REAL;
	reverseMoveRequired : BOOL;

END_VAR

//	Function Block: FB_SimMotor()
//	Description: A simulated motor axis to test MC commands
//
//	Created by: Ben Hess
//	Created Date: Tuesday, May 14th, 2019

homingTimer();
movingTimer();
resetTimer();
PowerState := PowerOn;
EnableState := DriveEnable;

IF AckError THEN
	_reset := TRUE;
END_IF

IF _reset THEN
	//Error := FALSE;
	resetTimer.IN := TRUE;
	HomingDone := FALSE;
	_reset := FALSE;
END_IF

IF resetTimer.Q THEN
	Error := FALSE;
	resetTimer.IN := FALSE;
END_IF

IF simFault THEN
	Error := TRUE;
	HomingDone := FALSE;
	simFault := FALSE;
	TargetReached := FALSE;
END_IF

CASE state OF
	0:		// Idle
			IF StartHoming THEN
				state := 1;
			END_IF

			IF MoveAbs THEN
				TargetReached := FALSE;
				IF TargetPosDist > ActPos THEN
					reverseMoveRequired := FALSE;
				ELSE
					reverseMoveRequired := TRUE;
				END_IF
				distanceToMove := ABS(ActPos - TargetPosDist);
				MoveAbs := FALSE;
				AxisState := Sharp_Motion.AXIS_STATE.AS_DiscreteMotion;
				state := 2;
			END_IF

			IF MoveRel THEN
				TargetReached := FALSE;
				distanceToMove := TargetPosDist;
				state := 2;
			END_IF

	1:		// Homing
			homingTimer.PT := T#5S;
			homingTimer.IN := TRUE;

			IF homingTimer.Q THEN
				homingTimer.IN := FALSE;
				ActPos := 2.0;
				HomingDone := TRUE;
				state := 100;
			END_IF

	2: 		// Moving to position
			movingTimer.PT := TO_TIME((distanceToMove * 1/ProfileVelocity) * 1000);
			movingTimer.IN := TRUE;
			IF reverseMoveRequired THEN
				ActPos := TargetPosDist - ((TO_REAL(movingTimer.ET) * ProfileVelocity)  / 1000) + distanceToMove;
			ELSE
				ActPos := TargetPosDist - ((TO_REAL(movingTimer.PT - movingTimer.ET) * ProfileVelocity)  / 1000);
			END_IF

			IF Halt THEN
				state := 100;
				AxisState := Sharp_Motion.AXIS_STATE.AS_Standstill;
			END_IF
			IF movingTimer.Q THEN
				movingTimer.IN := FALSE;
				TargetReached := TRUE;
				AxisState := Sharp_Motion.AXIS_STATE.AS_Standstill;
				state := 100;
			END_IF

	3:		//

	100:	// Clear/Reset
			homingTimer.IN := FALSE;
			movingTimer.IN := FALSE;

			state := 0;

END_CASE

FUNCTION_BLOCK FB_SimMotor EXTENDS Sharp_Motion.Axis_REF
VAR_INPUT
	simFault : BOOL;
END_VAR
VAR_OUTPUT
END_VAR
VAR
	homingTimer : Standard.TON;
	movingTimer : Standard.TON;
	resetTimer : Standard.TON := (PT := T#500ms);
	state : INT;
	homingState : INT;
	moveAbsState : INT;
	moveRelState : INT;
	_reset : BOOL;
	distanceToMove : REAL;
	reverseMoveRequired : BOOL;

END_VAR

//	Function Block: FB_SimMotor()
//	Description: A simulated motor axis to test MC commands
//
//	Created by: Ben Hess
//	Created Date: Tuesday, May 14th, 2019

homingTimer();
movingTimer();
resetTimer();
PowerState := PowerOn;
EnableState := DriveEnable;

IF AckError THEN
	_reset := TRUE;
END_IF

IF _reset THEN
	//Error := FALSE;
	resetTimer.IN := TRUE;
	HomingDone := FALSE;
	_reset := FALSE;
END_IF

IF resetTimer.Q THEN
	Error := FALSE;
	resetTimer.IN := FALSE;
END_IF

IF simFault THEN
	Error := TRUE;
	HomingDone := FALSE;
	simFault := FALSE;
	TargetReached := FALSE;
END_IF

CASE state OF
	0:		// Idle
			IF StartHoming THEN
				state := 1;
			END_IF

			IF MoveAbs THEN
				TargetReached := FALSE;
				IF TargetPosDist > ActPos THEN
					reverseMoveRequired := FALSE;
				ELSE
					reverseMoveRequired := TRUE;
				END_IF
				distanceToMove := ABS(ActPos - TargetPosDist);
				MoveAbs := FALSE;
				AxisState := Sharp_Motion.AXIS_STATE.AS_DiscreteMotion;
				state := 2;
			END_IF

			IF MoveRel THEN
				TargetReached := FALSE;
				distanceToMove := TargetPosDist;
				state := 2;
			END_IF

	1:		// Homing
			homingTimer.PT := T#5S;
			homingTimer.IN := TRUE;

			IF homingTimer.Q THEN
				homingTimer.IN := FALSE;
				ActPos := 2.0;
				HomingDone := TRUE;
				state := 100;
			END_IF

	2: 		// Moving to position
			movingTimer.PT := TO_TIME((distanceToMove * 1/ProfileVelocity) * 1000);
			movingTimer.IN := TRUE;
			IF reverseMoveRequired THEN
				ActPos := TargetPosDist - ((TO_REAL(movingTimer.ET) * ProfileVelocity)  / 1000) + distanceToMove;
			ELSE
				ActPos := TargetPosDist - ((TO_REAL(movingTimer.PT - movingTimer.ET) * ProfileVelocity)  / 1000);
			END_IF

			IF Halt THEN
				state := 100;
				AxisState := Sharp_Motion.AXIS_STATE.AS_Standstill;
			END_IF
			IF movingTimer.Q THEN
				movingTimer.IN := FALSE;
				TargetReached := TRUE;
				AxisState := Sharp_Motion.AXIS_STATE.AS_Standstill;
				state := 100;
			END_IF

	3:		//

	100:	// Clear/Reset
			homingTimer.IN := FALSE;
			movingTimer.IN := FALSE;

			state := 0;

END_CASE

(* ---- FB_SimMotor_UnitTests.st ---- *)
{attribute 'test' := 'multitest'}
{attribute 'testcasename':='Monostable Multivibrator'}
{attribute 'testcategory':='Basics'}
{attribute 'testcasetimeout':='360000'}

FUNCTION_BLOCK FB_SimMotor_UnitTests EXTENDS CBM.EtrigA
VAR_INPUT
	xGetTestInfo : BOOL;
    diTestCaseIndex : DINT;
END_VAR
VAR_OUTPUT
    sTestCaseName : STRING;
	sTestCaseCategories : STRING;
    diTestCaseCount : DINT;
    diTestCaseTimeout : DINT;
    sInfo : STRING;
	eError : UnitTestErrors;
    sError : STRING;
    eFailureMode : TM.FAILUREMODE;
END_VAR
VAR
	testee : FB_SimMotor();
	MC_MoveABSTestee : Sharp_Motion.MC_MoveAbsolute;
	MC_MoveABSTorqueTestee : Sharp_Motion.MC_MoveAbsoluteTorqueLimited;
	MC_MoveRELTestee : Sharp_Motion.MC_MoveRelative;
	MC_PowerTestee : Sharp_Motion.MC_Power;
	MC_HomeTestee : Sharp_Motion.MC_Home;
	delayTimer : Standard.TON;
END_VAR
SUPER^();

delayTimer();

testee();

MC_MoveABSTestee(Axis := testee);
MC_MoveABSTorqueTestee(Axis := testee);
MC_MoveRELTestee(Axis := testee);
MC_PowerTestee(Enable := TRUE, Axis := testee);
MC_HomeTestee(Axis := testee);

{attribute 'hide'}
METHOD prvAbort : BOOL

SUPER^.prvAbort();

xAbortInProgress := FALSE;

{attribute 'hide'}
METHOD prvCyclicAction : BOOL

SUPER^.prvCyclicAction();
MC_MoveRELTestee.Acceleration := 100;
MC_MoveRELTestee.Deceleration := 100;

CASE diTestCaseIndex OF
    0: 	IF THIS^.xGetTestInfo THEN
            THIS^.sTestCaseName := 'Step 1: Try to move motor before powering up';
            THIS^.sTestCaseCategories := 'General';
            THIS^.diTestCaseTimeout := 3000;
			xDone := TRUE;
		ELSE

			MC_MoveRELTestee.Velocity := 1;
			MC_MoveRELTestee.Distance := 5.6;
			MC_MoveRELTestee.Execute := TRUE;
			THIS^.RunTestFBs();

			IF testee.ActualPosition = 0
				AND MC_MoveRELTestee.Error
				AND MC_MoveRELTestee.ErrorID = Sharp_Motion.MC_ERROR.AXIS_NOT_READY
				THEN
				 xDone := TRUE;
			ELSE
				THIS^.sError := Standard.CONCAT('Axis did not error out ', CONCAT(TO_STRING(testee.ActualPosition),CONCAT(TO_STRING(MC_MoveRELTestee.Error), TO_STRING(MC_MoveRELTestee.ErrorID))));
				xError := TRUE;
				eError := UnitTestErrors.Failure;
            	eFailureMode := TM.FAILUREMODE.AbortTestCase;
                iError := 1;
			END_IF
        END_IF
    1: 	IF THIS^.xGetTestInfo THEN
            THIS^.sTestCaseName := 'Step 2: Power Up and move';
            THIS^.sTestCaseCategories := 'General';
            THIS^.diTestCaseTimeout := 15000;
			xDone := TRUE;
		ELSE
			MC_PowerTestee.RegulatorOn := TRUE;
			MC_PowerTestee.DriveStart := TRUE;
			RunTestFBs();
			MC_MoveRELTestee.Distance := 5.6;
			MC_MoveRELTestee.Execute := TRUE;
			delayTimer.PT := T#6S;
			delayTimer.IN := TRUE;

			IF delayTimer.Q THEN
				IF TO_DINT(testee.ActualPosition * 10) = 56 THEN
					xDone := TRUE;
				ELSE
					THIS^.sError := Standard.CONCAT('Axis did not move: Expected 5.6 got: ',TO_STRING(testee.ActualPosition));
					xError := TRUE;
					eError := UnitTestErrors.Failure;
					eFailureMode := TM.FAILUREMODE.AbortTestCase;
					iError := 1;
				END_IF
			END_IF

        END_IF

	2: 	IF THIS^.xGetTestInfo THEN
            THIS^.sTestCaseName := 'Step 3: ';
            THIS^.sTestCaseCategories := 'General';
            THIS^.diTestCaseTimeout := 3000;
			xDone := TRUE;
		ELSE
			(*TEST SOMETHING HERE*)
			IF (*CONNDITION*) FALSE THEN
				 xDone := TRUE;
			ELSE
				THIS^.sError := '';
				xError := TRUE;
				eError := UnitTestErrors.Failure;
            	eFailureMode := TM.FAILUREMODE.AbortTestCase;
                iError := 1;
			END_IF
        END_IF

   	3: 	IF THIS^.xGetTestInfo THEN
            THIS^.sTestCaseName := 'Step 4: ';
            THIS^.sTestCaseCategories := 'General';
            THIS^.diTestCaseTimeout := 3000;
			xDone := TRUE;
		ELSE
			(*TEST SOMETHING HERE*)
			IF (*CONNDITION*) FALSE THEN
				 xDone := TRUE;
			ELSE
				THIS^.sError := '';
				xError := TRUE;
				eError := UnitTestErrors.Failure;
            	eFailureMode := TM.FAILUREMODE.AbortTestCase;
                iError := 1;
			END_IF
        END_IF

	4: 	IF THIS^.xGetTestInfo THEN
            THIS^.sTestCaseName := 'Step 5: ';
            THIS^.sTestCaseCategories := 'General';
            THIS^.diTestCaseTimeout := 3000;
			xDone := TRUE;
		ELSE
			(*TEST SOMETHING HERE*)
			IF (*CONNDITION*) FALSE THEN
				 xDone := TRUE;
			ELSE
				THIS^.sError := '';
				xError := TRUE;
				eError := UnitTestErrors.Failure;
            	eFailureMode := TM.FAILUREMODE.AbortTestCase;
                iError := 1;
			END_IF
        END_IF

	5: 	IF THIS^.xGetTestInfo THEN
            THIS^.sTestCaseName := 'Step 6: ';
            THIS^.sTestCaseCategories := 'General';
            THIS^.diTestCaseTimeout := 3000;
			xDone := TRUE;
		ELSE
			(*TEST SOMETHING HERE*)
			IF (*CONNDITION*) FALSE THEN
				 xDone := TRUE;
			ELSE
				THIS^.sError := '';
				xError := TRUE;
				eError := UnitTestErrors.Failure;
            	eFailureMode := TM.FAILUREMODE.AbortTestCase;
                iError := 1;
			END_IF
        END_IF

	6: 	IF THIS^.xGetTestInfo THEN
            THIS^.sTestCaseName := 'Step 7: ';
            THIS^.sTestCaseCategories := 'General';
            THIS^.diTestCaseTimeout := 3000;
			xDone := TRUE;
		ELSE
			(*TEST SOMETHING HERE*)
			IF (*CONNDITION*) FALSE THEN
				 xDone := TRUE;
			ELSE
				THIS^.sError := '';
				xError := TRUE;
				eError := UnitTestErrors.Failure;
            	eFailureMode := TM.FAILUREMODE.AbortTestCase;
                iError := 1;
			END_IF
        END_IF
    ELSE
        IF THIS^.diTestCaseIndex < 0 THEN
            THIS^.diTestCaseCount := 2;
            xDone := TRUE;
        ELSE
            THIS^.sInfo := 'Invalid test case index';
            eError := UnitTestErrors.Failure;
			xError := TRUE;
        END_IF
END_CASE

{attribute 'hide'}
METHOD prvResetOutputs : BOOL

SUPER^.prvResetOutputs();

sTestCaseName := '';
sTestCaseCategories := '';
diTestCaseCount := 0;
diTestCaseTimeout := 0;
sInfo := '';
sError := '';
eFailureMode := TM.FAILUREMODE.AbortTestCase;

MC_MoveRELTestee.Execute := FALSE;

RunTestFBs();

{attribute 'hide'}
METHOD prvStart : BOOL

METHOD RunTestFBs
VAR_INPUT
END_VAR

testee();

MC_MoveABSTestee(Axis := testee);
MC_MoveABSTorqueTestee(Axis := testee);
MC_MoveRELTestee(Axis := testee);
MC_PowerTestee(Enable := TRUE, Axis := testee);
MC_HomeTestee(Axis := testee);

(* ---- FB_SimulatedFeedback.st ---- *)
FUNCTION_BLOCK FB_SimulatedFeedback EXTENDS FB_BaseObject
VAR_INPUT
	in : BOOL;			// Start of feedback (usually an output)
	simFeedbackFault : BOOL;	// Enable a feedback fault
	faultDelay : DINT;			// Delay for feedback fault
	minDelay : DINT;	//Minimum delay in mS
	maxDelay : DINT;	//Maximum delay in mS
END_VAR
VAR_OUTPUT
	Q : BOOL;
	fault : BOOL;
END_VAR
VAR
	inONS : FB_ONS();
	QONS : FB_ONS();
	_beginTimer : BOOL;
	randomDelay : DINT;
	delayTimer : Standard.TON;
END_VAR

//	Function Block: FB_SimulatedFeedback
//	Description: Meant to simulate a feedback based off an input with an additional option to simulate a failed feedback signal
//				 Can be used for testing or for creating "feedback" for components that lack a sensor
//
//	Usage: simPbarInFB(in := movePbarInOutput, minDelay := 100, maxDelay := 200);
//
//	Created by: Ben Hess
//	Created Date: 3-2019

inONS(CLK := in);
QONS(CLK := Q);
IF minDelay < 0 THEN
	minDelay := 0;
END_IF
IF inONS.OSR THEN
	_logger.AddLogItem(CONCAT(_prefix,'Started'));
	// Feeback can be set as a range to simulate variations in air pressure, friction etc.
	// Choose a random delay in between min and max
	IF NOT simFeedbackFault THEN
		randomDelay := 	FN_RandomDINT(last := randomDelay,
								low := minDelay,
								high := maxDelay);
		delayTimer.PT := DINT_TO_TIME(randomDelay);
	ELSE
		// Use fault timer if fault sim enabled
		delayTimer.PT := DINT_TO_TIME(faultDelay);
	END_IF
END_IF

IF QONS.OSR AND NOT simFeedbackFault THEN
	_logger.AddLogItem(CONCAT(_prefix,'Done'));
END_IF

delayTimer(IN := in);

IF NOT simFeedbackFault THEN
	Q := delayTimer.Q;
	fault := FALSE;
ELSE
	Q := FALSE;
	fault := delayTimer.Q;
END_IF

(* ---- FB_SimulatedFeedbackPhysicalInput.st ---- *)
FUNCTION_BLOCK FB_SimulatedFeedbackPhysicalInput EXTENDS FB_SimulatedFeedback
VAR_INPUT
	inputToSimulate : REFERENCE TO FB_PhysicalDigitalInput;
END_VAR
VAR_OUTPUT

END_VAR
VAR

END_VAR

//	Function Block: FB_SimulatedFeedbackPhysicalInput
//	Description: Meant to simulate a feedback based off an input with an additional option to simulate a failed feedback signal
//				 Using a physical input to simulate
//
//	Usage: simPbarInFB(in := movePbarInOutput, minDelay := 100, maxDelay := 200);
//
//	Created by: Ben Hess
//	Created Date: 5-20-2019

SUPER^();

IF inputToSimulate.simulate = TRUE THEN
	inputToSimulate.simValue := Q;
END_IF

(* ---- FB_Simulation.st ---- *)
{attribute 'FBVisuCreator'}
FUNCTION_BLOCK FB_Simulation
VAR_INPUT
	failedToGrabBagLeftFinger : BOOL;
	failedToGrabBagRightFinger : BOOL;
	failedToGrabBagBothFingers : BOOL;
	pressureBarFailedToMoveIn : BOOL;
	pressureBarFailedToMoveOut : BOOL;
	pressureBarObstucted : BOOL;
	pressureBarfailedToHome : BOOL;
	passthroughMotorFault : BOOL;
	failedToMovePassthrough : BOOL;
	msfHorizontalFailedToHome : BOOL;
END_VAR
VAR_OUTPUT
END_VAR
VAR
END_VAR

(* ---- FB_SingleSolenoidNormallyRetractedActuator.st ---- *)
FUNCTION_BLOCK FB_SingleSolenoidNormallyRetractedActuator EXTENDS FB_PneumaticActuator IMPLEMENTS ICylinder
VAR_INPUT
END_VAR
VAR_OUTPUT
END_VAR
VAR
END_VAR

PROPERTY ExtendAsserted : BOOL

PROPERTY RetractAsserted : BOOL

METHOD Extend

solenoid0 := TRUE;

METHOD Retract

solenoid0 := FALSE;

(* ---- FB_SingleSolenoidNormallyRetractedActuator_UnitTests.st ---- *)
(*
*)
{attribute 'test' := 'multitest'}
{attribute 'testcasename':='Single Solenoid Normally Retracted'}
{attribute 'testcategory':='Solenoids'}
{attribute 'testcasetimeout':='15000'}
FUNCTION_BLOCK FB_SingleSolenoidNormallyRetractedActuator_UnitTests EXTENDS CBM.EtrigA
VAR_INPUT
	xGetTestInfo : BOOL;
    diTestCaseIndex : DINT;
END_VAR
VAR_OUTPUT
    sTestCaseName : STRING;
	sTestCaseCategories : STRING;
    diTestCaseCount : DINT;
    diTestCaseTimeout : DINT;
    sInfo : STRING;
	eError : UnitTestErrors;
    sError : STRING;
    eFailureMode : TM.FAILUREMODE;
END_VAR
VAR
	testee : FB_SingleSolenoidNormallyRetractedActuator(name := 'Unit Test Actuator');
END_VAR
SUPER^();

{attribute 'hide'}
METHOD prvAbort : BOOL

SUPER^.prvAbort();

xAbortInProgress := FALSE;

{attribute 'hide'}
METHOD prvCyclicAction : BOOL

SUPER^.prvCyclicAction();
THIS^.diTestCaseCount := 3;

CASE diTestCaseIndex OF
    0: // Test Case #0
        IF THIS^.xGetTestInfo THEN
            THIS^.sTestCaseName := 'Step 1: Test Solonoids Off';
            THIS^.sTestCaseCategories := 'Solenoids';
            THIS^.diTestCaseTimeout := 3000;
			xDone := TRUE;
		ELSE
			IF NOT testee.Solenoid0Asserted AND NOT testee.Solenoid1Asserted AND testee.RetractAsserted THEN
				 xDone := TRUE;
			ELSE
				THIS^.sError := 'Solenoids not off';
				xError := TRUE;
				eError := UnitTestErrors.Failure;
            	eFailureMode := TM.FAILUREMODE.AbortTestCase;
                iError := 1;
			END_IF
        END_IF
    1: // Test Case #1
        IF THIS^.xGetTestInfo THEN
            THIS^.sTestCaseName := 'Step 2: Extend Cylinder';
            THIS^.sTestCaseCategories := 'Solenoids';
            THIS^.diTestCaseTimeout := 3000;
            xDone := TRUE;
		ELSE
			testee.Extend();
			IF testee.Solenoid0Asserted AND testee.ExtendAsserted
				AND NOT testee.Solenoid1Asserted AND NOT testee.RetractAsserted THEN
				 xDone := TRUE;
			ELSE
				THIS^.sError := 'Failed to extend';
				xError := TRUE;
				eError := UnitTestErrors.Failure;
            	eFailureMode := TM.FAILUREMODE.AbortTestCase;
                iError := 2;
			END_IF
       END_IF

	2:	//
		IF THIS^.xGetTestInfo THEN
            THIS^.sTestCaseName := 'Step 3: Retract Cylinder';
            THIS^.sTestCaseCategories := 'Solenoids';
            THIS^.diTestCaseTimeout := 3000;
            xDone := TRUE;
		ELSE
			testee.Retract();
			IF NOT testee.Solenoid0Asserted AND NOT testee.ExtendAsserted AND testee.RetractAsserted THEN
				 xDone := TRUE;
			ELSE
				THIS^.sError := 'Failed to retract';
				xError := TRUE;
				eError := UnitTestErrors.Failure;
            	eFailureMode := TM.FAILUREMODE.AbortTestCase;
                iError := 3;
			END_IF
       END_IF
    ELSE
        IF THIS^.diTestCaseIndex < 0 THEN
            THIS^.diTestCaseCount := 3;
            xDone := TRUE;
        ELSE
            THIS^.sInfo := 'Invalid test case index';
            eError := UnitTestErrors.Failure;
			xError := TRUE;
        END_IF
END_CASE

{attribute 'hide'}
METHOD prvResetOutputs : BOOL

SUPER^.prvResetOutputs();

sTestCaseName := '';
sTestCaseCategories := '';
diTestCaseCount := 0;
diTestCaseTimeout := 0;
sInfo := '';
sError := '';
eFailureMode := TM.FAILUREMODE.AbortTestCase;

{attribute 'hide'}
METHOD prvStart : BOOL

SUPER^.prvStart();

(* ---- FB_SolenoidValve.st ---- *)
FUNCTION_BLOCK FB_SolenoidValve EXTENDS FB_BaseObject IMPLEMENTS ISolenoidValve, ISimulateable
VAR_INPUT

END_VAR
VAR_OUTPUT
	solenoid0 : BOOL;
	solenoid1 : BOOL;
END_VAR
VAR
	_simulateActive : BOOL;
END_VAR

PROPERTY Simulate : BOOL

PROPERTY Solenoid0Asserted : BOOL

PROPERTY Solenoid1Asserted : BOOL

FUNCTION_BLOCK FB_SolenoidValve EXTENDS FB_BaseObject IMPLEMENTS ISolenoidValve, ISimulateable
VAR_INPUT

END_VAR
VAR_OUTPUT
	solenoid0 : BOOL;
	solenoid1 : BOOL;
END_VAR
VAR
	_simulateActive : BOOL;
END_VAR

PROPERTY Simulate : BOOL

PROPERTY Solenoid0Asserted : BOOL

PROPERTY Solenoid1Asserted : BOOL

(* ---- FB_SolenoidValveManifold.st ---- *)
FUNCTION_BLOCK FB_SolenoidValveManifold EXTENDS FB_BaseObject
VAR_INPUT
	ptrEIPOutputs : POINTER TO DWORD;	// Pointer to starting word of EIP Outputs for the I/O Image

	station : ARRAY[1..16] OF ISolenoidValve;	// Array of up to 16 valve stations on manifold

END_VAR
VAR_OUTPUT
END_VAR
VAR
	i : INT;
	j : INT;
END_VAR

//	Function Block: FB_SolenoidValveManifold
//	Description: Sets the output image of the valve manifold (ptrEIPOutputs) to the correct values depending on configuration.
//
//	Usage: All stations should be configured with a valve before running.
//
//	Created by: Ben Hess
//	Created Date: 6-27-2019

// Loop through all possible stations
FOR i := 1 TO 16 DO
	IF station[i] <> 0 THEN	// Check for valid reference passed into the station interface
		// If ref good then set I/O image bit for proper station.  If simulated then don't set real output for solenoid
		ptrEIPOutputs^ := OSCAT_BASIC.BIT_LOAD_DW(in := ptrEIPOutputs^, POS := j, VAL := station[i].Solenoid0Asserted AND NOT station[i].Simulate);
		ptrEIPOutputs^ := OSCAT_BASIC.BIT_LOAD_DW(in := ptrEIPOutputs^, POS := j+1, VAL := station[i].Solenoid1Asserted AND NOT station[i].Simulate);
	END_IF
	j := j + 2;
END_FOR
// Restart bit loop
j := 0;

FUNCTION_BLOCK FB_SolenoidValveManifold EXTENDS FB_BaseObject
VAR_INPUT
	ptrEIPOutputs : POINTER TO DWORD;	// Pointer to starting word of EIP Outputs for the I/O Image

	station : ARRAY[1..16] OF ISolenoidValve;	// Array of up to 16 valve stations on manifold

END_VAR
VAR_OUTPUT
END_VAR
VAR
	i : INT;
	j : INT;
END_VAR

//	Function Block: FB_SolenoidValveManifold
//	Description: Sets the output image of the valve manifold (ptrEIPOutputs) to the correct values depending on configuration.
//
//	Usage: All stations should be configured with a valve before running.
//
//	Created by: Ben Hess
//	Created Date: 6-27-2019

// Loop through all possible stations
FOR i := 1 TO 16 DO
	IF station[i] <> 0 THEN	// Check for valid reference passed into the station interface
		// If ref good then set I/O image bit for proper station.  If simulated then don't set real output for solenoid
		ptrEIPOutputs^ := OSCAT_BASIC.BIT_LOAD_DW(in := ptrEIPOutputs^, POS := j, VAL := station[i].Solenoid0Asserted AND NOT station[i].Simulate);
		ptrEIPOutputs^ := OSCAT_BASIC.BIT_LOAD_DW(in := ptrEIPOutputs^, POS := j+1, VAL := station[i].Solenoid1Asserted AND NOT station[i].Simulate);
	END_IF
	j := j + 2;
END_FOR
// Restart bit loop
j := 0;
